// TIA Portal V17 program export: 3 tag tables, 8 data types, 18 data blocks, 27 code blocks (in call order from the OBs), 10 instance data blocks

VAR_GLOBAL   // PLC tag table "Customer"
   "VB3-M8301 Start" AT %I200.0 : Bool;   // Anfrage starten 1 = Wärmepumpe starten, 0 = nichts tun
   "VB3-M8301 Stop" AT %I200.1 : Bool;   // Stopp-Anfrage 1 = stoppen, 0 = nichts tun (überschreibt das Startsignal)
   "VB3-M8301 Freigabe" AT %I200.2 : Bool;   // Freigabe 1 = Startbefehl aktivieren 0 = Startbefehl ignorieren
   "VB3-M8301 Reset" AT %I200.3 : Bool;   // Alarmbestätigung 1 = alle Alarme löschen, 0 = nichts tun
   "VB3-M8301 Not-Aus" AT %I200.4 : Bool;   // Not-Aus zurücksetzen 1 = Not-Aus zurücksetzen, 0 = nichts tun
   "VB3-M8301 Sstop" AT %I200.5 : Bool;   // Schnellstopp-Anfrage 1 = Schnellstoppanforderung, 0 = nichts tun
   "A1024.6" AT %I200.6 : Bool;   // Reserve
   "A1024.7" AT %I200.7 : Bool;   // Reserve
   QI117_828B2 AT %I203.0 : Bool;   // Rückmeldung zur Raumlüftung WP1 1 = Lüftung ok, 0 = Startbefehl ignorieren
   QI117_828B3 AT %I203.1 : Bool;   // Kondensierbare Gase erkannt WP1 1 = Anforderung stoppen und Absperrventile schließen, 0 = nichts tun
   "A1027.2" AT %I203.2 : Bool;   // Reserve
   "A1027.3" AT %I203.3 : Bool;   // Reserve
   "A1027.4" AT %I203.4 : Bool;   // Reserve
   "A1027.5" AT %I203.5 : Bool;   // Reserve
   "A1027.6" AT %I203.6 : Bool;   // Reserve
   "VB3-M8301 Live bit" AT %I203.7 : Bool;   // Live bit
   QI117_828B1 AT %IW201 : Int;   // [%] Leistungssollwert WP1 Sollwert für die Systemleistung
   AW1028 AT %IW204 : Int;   // Reserve
   AW1030 AT %IW206 : Int;   // Reserve
   "VB3-M8301 NA-Status" AT %Q200.0 : Bool;   // Not-Aus-Status 1 = Not-Aus ok, 0 = Not-Aus aktiv
   "VB3-M8301 G1 Ein" AT %Q200.1 : Bool;   // Status der Ölheizungen Gruppe 1 1 = Heizungen ein, 0 = Heizungen aus
   "VB3-M8301 G2 Ein" AT %Q200.2 : Bool;   // Status der Ölheizungen Gruppe 2 1 = Heizungen ein, 0 = Heizungen aus
   "E1024.3" AT %Q200.3 : Bool;   // Reserve
   "E1024.4" AT %Q200.4 : Bool;   // Reserve
   "E1024.5" AT %Q200.5 : Bool;   // Reserve
   "E1024.6" AT %Q200.6 : Bool;   // Reserve
   "E1024.7" AT %Q200.7 : Bool;   // Reserve
   GH117_827 AT %Q201.0 : Bool;   // Absalzventil 1 = offen, 0 = geschlossen, gesteuert durch Heaten
   GH117_826_1 AT %Q201.1 : Bool;   // Ventil nicht kondensierbares Gase 1 1 = offen, 0 = geschlossen, gesteuert durch Heaten
   GH117_826_2 AT %Q201.2 : Bool;   // Ventil nicht kondensierbares Gase 2 1 = offen, 0 = geschlossen, gesteuert durch Heaten
   "E1025.3" AT %Q201.3 : Bool;   // Reserve
   "E1025.4" AT %Q201.4 : Bool;   // Reserve
   "E1025.5" AT %Q201.5 : Bool;   // Reserve
   "E1025.6" AT %Q201.6 : Bool;   // Reserve
   "E1025.7 Live Bit" AT %Q201.7 : Bool;   // Live bit
   "VB3-M8301 Status" AT %QW202 : Int;   // Maschinenzustand 0 = Initialisierung, 1 = Offline, 2 = Standby, Aufwärmen, Betrieb usw. (Aufzählungstyp)
   QI117_828B4 AT %QW204 : Int;   // [h] Betriebsstunden Zählt, solange der Heatbooster eingeschaltet ist
   QI117_828B5 AT %QW206 : Int;   // [h] Aktive Zeit Stunden Aktiv bedeutet, dass die Maschine eingeschaltet ist (entweder im Betrieb oder im Leerlauf).
   QI117_828B6 AT %QW208 : Int;   // [h] Laufzeit Stunden Laufen bedeutet in Betrieb (Wärmeerhöhung!)
   QI117_828B7 AT %QW210 : Int;   // [C] HBL-TT-07 (HBL-TT-901) Temperatur Saugseite Kondensator
   QI117_828B8 AT %QW212 : Int;   // [C] HBL-TT-08 (HBL-TT-518) Temperatur Druckseit Kondensator
   QI117_828B9 AT %QW214 : Int;   // [C] HBL-TT-13 (HBL-TT-546) Temperatur Saugseite Verdampfer
   QI117_828B10 AT %QW216 : Int;   // [C] HBL-TT-14 (HBL-TT-542) Temperatur Druckseit Verdampfer
   QI117_828B11 AT %QW218 : Int;   // [C] HBL-TT-16 Lufttemperatur des Containers
   QI117_828B12 AT %QW220 : Int;   // [C] HBL-TT-17 Lufttemperatur im Schaltschrank
   QI117_828B13 AT %QW222 : Int;   // [C] HBL-TT-18 Umgebungslufttemperatur
   QI117_828B16 AT %QW224 : Int;   // [ppm] HBL-CT-03 Gasdetektor Container
   QI117_828B17 AT %QW226 : Int;   // [%] SSC-LT-01 Füllstand des Sperrflüssigkeitsbehälters
   "VB3-M8301 Wärme" AT %QW228 : Int;   // [kW] Voraussichtliche Wärmelieferung
   QI117_828B18 AT %QW230 : Int;   // [1] System: COP
   "VB3-M8301 kW" AT %QW232 : Int;   // [kW] System: electrical power
   QI117_828B19 AT %QW234 : Int;   // [C] System: temperature lift
   GH117_812 AT %QW236 : Int;   // [%] Kondensatventil Verdampfer ein
   GH117_818 AT %QW238 : Int;   // [%] Dampfventil Verdampfer aus (HBL-HCV-514)
   GH117_815 AT %QW240 : Int;   // [%] Dampfventil Kondensator ein (HBL-HCV-548)
   GH117_821 AT %QW242 : Int;   // [%] Kondensatventil Kondensator aus
   EW1072 AT %QW248 : Int;   // Reserve
   "VB3-M8301 kW(1)" AT %QW244 : Int;   // Elektrische Leistung
   EW1070 AT %QW246 : Int;   // Reserve
   EW1074 AT %QW250 : Int;   // Reserve
END_VAR

VAR_GLOBAL   // PLC tag table "Default tag table"
   Clock_Byte AT %MB0 : Byte;
   Clock_10Hz AT %M0.0 : Bool;
   Clock_5Hz AT %M0.1 : Bool;
   "Clock_2.5Hz" AT %M0.2 : Bool;
   Clock_2Hz AT %M0.3 : Bool;
   "Clock_1.25Hz" AT %M0.4 : Bool;
   Clock_1Hz AT %M0.5 : Bool;
   "Clock_0.625Hz" AT %M0.6 : Bool;
   "Clock_0.5Hz" AT %M0.7 : Bool;
END_VAR

VAR_GLOBAL   // PLC tag table "Local_IO"
   DQa_0 AT %Q0.0 : Bool;
   DQa_1 AT %Q0.1 : Bool;
   DQa_2 AT %Q0.2 : Bool;
   DQa_3 AT %Q0.3 : Bool;
   DQa_4 AT %Q0.4 : Bool;
   DQa_5 AT %Q0.5 : Bool;
   DQa_6 AT %Q0.6 : Bool;
   DQa_7 AT %Q0.7 : Bool;
   DQb_0 AT %Q1.0 : Bool;
   DQb_1 AT %Q1.1 : Bool;
   DIa_0 AT %I0.0 : Bool;
   DIa_1 AT %I0.1 : Bool;
   DIa_2 AT %I0.2 : Bool;
   DIa_3 AT %I0.3 : Bool;
   DIa_4 AT %I0.4 : Bool;
   DIa_5 AT %I0.5 : Bool;
   DIa_6 AT %I0.6 : Bool;
   DIa_7 AT %I0.7 : Bool;
   DIb_0 AT %I1.0 : Bool;
   DIb_1 AT %I1.1 : Bool;
   DIb_2 AT %I1.2 : Bool;
   DIb_3 AT %I1.3 : Bool;
   DIb_4 AT %I1.4 : Bool;
   DIb_5 AT %I1.5 : Bool;
END_VAR

TYPE "stAnalogInput"
// stored: IsFailsafeCompliant false
   STRUCT
      Raw : "stRawValue";   // Raw values
      Eng : "stCalcValue";   // Engineering values
      bInitCmd : Bool;   // Recalculate scaling parameters
   END_STRUCT;
END_TYPE

TYPE "stAnalogOutput"
// stored: IsFailsafeCompliant false
   STRUCT
      Raw : "stRawValue";
      Eng { S7_SetPoint := 'True'} : "stCalcValue";
   END_STRUCT;
END_TYPE

TYPE "stCalcValue"
// stored: IsFailsafeCompliant false
   STRUCT
      fMin : Real;   // Negative-most value
      fMax : Real;   // Positive-most value
      fValue : Real;   // Actual value
      bError : Bool;   // Value invalid or out of range
      bCheckLimits : Bool := false;   // 1 = set bError if outside min & max, 0 = do nothing
      bLimited : Bool;   // 1 = value is limited, 0 = value is not limited
   END_STRUCT;
END_TYPE

TYPE "stHeartbeatCount2"
// stored: IsFailsafeCompliant false
   STRUCT
      nLocalCount : UInt;   // Count sent to remote partner
      nRemoteCount : UInt;   // Count received from remote partner
      bEnable : Bool;   // 1 = run heartbeat, 0 = disabled
      bOk : Bool;   // 1 = heatbeat ok, 0 = timeout
      nState : USInt;   // 0 = idle, 1 = ping, 2 = wait for pong, 3 = timeout
      tTimeout : Time := T#2s;   // Comm error timeout
   END_STRUCT;
END_TYPE

TYPE "stRawValue"
// stored: IsFailsafeCompliant false
   STRUCT
      iMin : Int;   // Module output at minimum input
      iMax : Int;   // Module output at maximum input
      iValue : Int;   // Current module value
      bFault : Bool;   // 0 = valid data, 1 = invalid data
   END_STRUCT;
END_TYPE

TYPE "stRegulatingValve"
// stored: IsFailsafeCompliant false
   STRUCT
      Cmd : Struct
         bManualMode : Bool;   // 1 = Manual Mode
         fManualValue : Real;   // manual position
         fOffset : Real;   // zero position offset
         Position : "stAnalogOutput";
      END_STRUCT;
      Stat : Struct
         Position : "stAnalogInput";
      END_STRUCT;
   END_STRUCT;
END_TYPE

TYPE "typeDataPtr"
// stored: IsFailsafeCompliant false
   STRUCT
      data : Array[0..7] of Word;
   END_STRUCT;
END_TYPE

TYPE "CAN-IDs_ToSend"
// stored: IsFailsafeCompliant false
   STRUCT
      IDs : Array[0..74] of Int;
   END_STRUCT;
   // IDs[0] := 16#0201;
   // IDs[1] := 16#0202;
   // IDs[2] := 16#0203;
   // IDs[3] := 16#0204;
   // IDs[4] := 16#0205;
   // IDs[5] := 16#0206;
   // IDs[6] := 16#0207;
   // IDs[7] := 16#0210;
   // IDs[8] := 16#0220;
   // IDs[9] := 16#0221;
   // IDs[10] := 16#0222;
   // IDs[11] := 16#0223;
   // IDs[12] := 16#0224;
   // IDs[13] := 16#0240;
   // IDs[14] := 16#0241;
   // IDs[15] := 16#0242;
   // IDs[16] := 16#0243;
   // IDs[17] := 16#0501;
   // IDs[18] := 16#0244;
   // IDs[19] := 16#0245;
   // IDs[20] := 16#0246;
   // IDs[21] := 16#0250;
   // IDs[22] := 16#0251;
   // IDs[23] := 16#0252;
   // IDs[24] := 16#0253;
   // IDs[25] := 16#0254;
   // IDs[26] := 16#0260;
   // IDs[27] := 16#0261;
   // IDs[28] := 16#0262;
   // IDs[29] := 16#0263;
   // IDs[30] := 16#0264;
   // IDs[31] := 16#0301;
   // IDs[32] := 16#0302;
   // IDs[33] := 16#0310;
   // IDs[34] := 16#0311;
   // IDs[35] := 16#0312;
   // IDs[36] := 16#0313;
   // IDs[37] := 16#0314;
   // IDs[38] := 16#0320;
   // IDs[39] := 16#0321;
   // IDs[40] := 16#0322;
   // IDs[41] := 16#0323;
   // IDs[42] := 16#0324;
   // IDs[43] := 16#0241;
   // IDs[44] := 16#0243;
   // IDs[45] := 16#0501;
   // IDs[46] := 16#0401;
   // IDs[47] := 16#0402;
   // IDs[48] := 16#0403;
   // IDs[49] := 16#0404;
   // IDs[50] := 16#0405;
   // IDs[51] := 16#0451;
   // IDs[52] := 16#0452;
   // IDs[53] := 16#0453;
   // IDs[54] := 16#0454;
   // IDs[55] := 16#0455;
   // IDs[56] := 16#0456;
   // IDs[57] := 16#0457;
   // IDs[58] := 16#0458;
   // IDs[59] := 16#0459;
   // IDs[60] := 16#0460;
END_TYPE

DATA_BLOCK "DB_AI"   // DB40
{ S7_Optimized_Access := 'FALSE' }
AUTHOR : Heaten
VERSION : 0.1
// stored: AutoNumber true, DBAccessibleFromOPCUA true, IsOnlyStoredInLoadMemory false, IsWriteProtectedInAS false
   VAR RETAIN
      Dummy : Bool;   // All locally-connected AIs go here
   END_VAR
BEGIN
END_DATA_BLOCK

DATA_BLOCK "DB_Calc"   // DB45
{ S7_Optimized_Access := 'FALSE' }
VERSION : 0.1
// stored: AutoNumber true, DBAccessibleFromOPCUA true, IsOnlyStoredInLoadMemory false, IsWriteProtectedInAS false
   VAR
      Dummy : Bool;   // Locally calculated values go here
   END_VAR
BEGIN
END_DATA_BLOCK

DATA_BLOCK "DB_CurrentSetting"   // DB21
{ S7_Optimized_Access := 'TRUE' }
AUTHOR : Heaten
VERSION : 0.1
// stored: AutoNumber false, DBAccessibleFromOPCUA true, IsOnlyStoredInLoadMemory false, IsRetainMemResEnabled false, IsWriteProtectedInAS false, MemoryReserve 0
   VAR RETAIN
      HeatSourceFlowLimit : Real := 0.0;   // [L/s] Heat source minimum volume flow
      HeatSinkFlowLimit : Real := 0.0;   // [L/s] Heat sink minimum volume flow
      "CAN-ModuleActive" : Bool := TRUE;   // 1 = do CAN comm, 0 = skip it
   END_VAR
BEGIN
END_DATA_BLOCK

DATA_BLOCK "DB_Customer"   // DB10
{ S7_Optimized_Access := 'TRUE' }
AUTHOR : Heaten
VERSION : 0.1
// stored: AutoNumber true, DBAccessibleFromOPCUA true, IsOnlyStoredInLoadMemory false, IsRetainMemResEnabled false, IsWriteProtectedInAS false, MemoryReserve 100
   VAR
      bEnabled : Bool;   // Enable Customer interface
      Watchdog : "stHeartbeatCount2";   // Comm monitoring Customer <-> Heatbooster
      Dummy { S7_SetPoint := 'True'} : "stCalcValue";
   END_VAR
BEGIN
END_DATA_BLOCK

DATA_BLOCK "DB_DI"   // DB2
{ S7_Optimized_Access := 'TRUE' }
VERSION : 0.1
// stored: AutoNumber false, DBAccessibleFromOPCUA true, IsOnlyStoredInLoadMemory false, IsRetainMemResEnabled false, IsWriteProtectedInAS false, MemoryReserve 0
   VAR
      EXT_FS_01 : Bool;   // Flow switch heat source (local)
      EXT_FS_02 : Bool;   // Flow switch heat sink (local)
   END_VAR
BEGIN
END_DATA_BLOCK

DATA_BLOCK "DB_DO"   // DB8
{ S7_Optimized_Access := 'TRUE' }
VERSION : 0.1
// stored: AutoNumber false, DBAccessibleFromOPCUA true, IsOnlyStoredInLoadMemory false, IsRetainMemResEnabled false, IsWriteProtectedInAS false, MemoryReserve 100
   VAR
      HBL_EC_01 : Bool;
      HBL_EC_02 : Bool;
      HBL_HV_630 : Bool;
      HBL_HV_114 : Bool;
      HBL_HV_115 : Bool;
      HBL_HV_860 : Bool;
      HBL_HV_861 : Bool;
      HBL_XV_06 : Bool;
      HBL_XV_07 : Bool;
      HBL_HV_631 : Bool;
      SSC_P_01 : Bool;
      SSC_F_01 : Bool;
      SSC_P_02 : Bool;
      CPC_P_01 : Bool;
      GH117_827 : Bool;   // Blowdown valve
      GH117_826_1 : Bool;   // NCG valve 1
      GH117_826_2 : Bool;   // NCG valve 2
      HBL_LSH_62 : Bool;
      HBL_LSL_63 : Bool;
      HBL_LSH_64 : Bool;
      HBL_LSL_864 : Bool;
      HBL_LS_632 : Bool;
      HBL_LS_633 : Bool;
   END_VAR
BEGIN
END_DATA_BLOCK

DATA_BLOCK "DB_Heatbooster"   // DB19
{ S7_Optimized_Access := 'TRUE' }
VERSION : 0.1
// stored: AutoNumber true, DBAccessibleFromOPCUA true, IsOnlyStoredInLoadMemory false, IsRetainMemResEnabled false, IsWriteProtectedInAS false, MemoryReserve 0
   VAR
      AI : Struct
         HBL_TT_502 { S7_SetPoint := 'True'} : "stCalcValue";   // Compressor discharge popoff temperature
         HBL_PT_503 { S7_SetPoint := 'True'} : "stCalcValue";   // Compressor discharge pressure
         HBL_TT_504 { S7_SetPoint := 'True'} : "stCalcValue";   // Compressor discharge temperature
         HBL_LT_510 { S7_SetPoint := 'True'} : "stCalcValue";   // Steam generator condensate level
         HBL_PT_511 { S7_SetPoint := 'True'} : "stCalcValue";   // Heat sink discharge pressure
         HBL_TT_512 { S7_SetPoint := 'True'} : "stCalcValue";   // Heat sink discharge temperature
         HBL_TT_516 { S7_SetPoint := 'True'} : "stCalcValue";   // Steam generator suction temperature
         HBL_PT_517 { S7_SetPoint := 'True'} : "stCalcValue";   // Steam generator suction pressure
         HBL_TT_518 { S7_SetPoint := 'True'} : "stCalcValue";   // Heat sink discharge process temperature
         HBL_PT_519 { S7_SetPoint := 'True'} : "stCalcValue";   // Heat sink discharge process pressure
         HBL_FT_520 { S7_SetPoint := 'True'} : "stCalcValue";   // Refrigerant flow
         HBL_TT_530 { S7_SetPoint := 'True'} : "stCalcValue";   // Expansion valve B discharge temperature
         HBL_PT_531 { S7_SetPoint := 'True'} : "stCalcValue";   // Expansion valve B discharge pressure
         HBL_TT_532 { S7_SetPoint := 'True'} : "stCalcValue";   // Heat source discharge B temperature
         HBL_TT_533 { S7_SetPoint := 'True'} : "stCalcValue";   // Evaporator B discharge temperature
         HBL_PT_534 { S7_SetPoint := 'True'} : "stCalcValue";   // Evaporator B discharge pressure
         HBL_AT_535 { S7_SetPoint := 'True'} : "stCalcValue";   // Evaporator B steam quality
         HBL_TT_540 { S7_SetPoint := 'True'} : "stCalcValue";   // Expansion valve A discharge temperature
         HBL_PT_541 { S7_SetPoint := 'True'} : "stCalcValue";   // Expansion valve A discharge pressure
         HBL_TT_542 { S7_SetPoint := 'True'} : "stCalcValue";   // Heat source discharge temperature
         HBL_TT_543 { S7_SetPoint := 'True'} : "stCalcValue";   // Evaporator A discharge temperature
         HBL_PT_544 { S7_SetPoint := 'True'} : "stCalcValue";   // Evaporator A discharge pressure
         HBL_AT_545 { S7_SetPoint := 'True'} : "stCalcValue";   // Evaporator A steam quality
         HBL_TT_546 { S7_SetPoint := 'True'} : "stCalcValue";   // Heat source suction temperature
         HBL_PT_547 { S7_SetPoint := 'True'} : "stCalcValue";   // Heast source suction pressure
         HBL_TT_571 { S7_SetPoint := 'True'} : "stCalcValue";   // Compressor suction temperature
         HBL_PT_572 { S7_SetPoint := 'True'} : "stCalcValue";   // Compressor suction pressure
         HBL_TT_573 { S7_SetPoint := 'True'} : "stCalcValue";   // Expansion valve suction temperature
         HBL_LT_610 { S7_SetPoint := 'True'} : "stCalcValue";   // HP receiver refrigerant level
         HBL_TT_611 { S7_SetPoint := 'True'} : "stCalcValue";   // Steam generator discharge temperature
         HBL_PT_612 { S7_SetPoint := 'True'} : "stCalcValue";   // Steam generator discharge pressure
         HBL_CT_615 { S7_SetPoint := 'True'} : "stCalcValue";   // Gas detector PSV discharge pipe
         HBL_PT_618 { S7_SetPoint := 'True'} : "stCalcValue";   // HP Receiver pressure
         HBL_PT_635 { S7_SetPoint := 'True'} : "stCalcValue";   // Oil separator stage 1 oil return pressure
         HBL_PT_636 { S7_SetPoint := 'True'} : "stCalcValue";   // Oil separator stage 2 oil return pressure
         HBL_LT_650 { S7_SetPoint := 'True'} : "stCalcValue";   // Heat source condensate buffer tank level
         HBL_PT_651 { S7_SetPoint := 'True'} : "stCalcValue";   // Heat source condensate buffer tank pressure
         HBL_PT_701 { S7_SetPoint := 'True'} : "stCalcValue";   // Filter dryer suction pressure
         HBL_PT_702 { S7_SetPoint := 'True'} : "stCalcValue";   // Filter dryer discharge pressure
         HBL_PT_703 { S7_SetPoint := 'True'} : "stCalcValue";   // Filter dryer differential pressure
         CPC_LT_870 { S7_SetPoint := 'True'} : "stCalcValue";   // CPC tank refrigerant level
         CPC_TT_871 { S7_SetPoint := 'True'} : "stCalcValue";   // CPC tank refrigerant temperature
         CPC_PT_872 { S7_SetPoint := 'True'} : "stCalcValue";   // CPC tank refrigerant pressure
         CPC_PT_862 { S7_SetPoint := 'True'} : "stCalcValue";   // CPC pump discharge pressure
         HBL_TT_901 { S7_SetPoint := 'True'} : "stCalcValue";   // Heat sink suction temperature
         HBL_PT_902 { S7_SetPoint := 'True'} : "stCalcValue";   // Heat sink suction pressure
         HBL_TT_03 { S7_SetPoint := 'True'} : "stCalcValue";   // Oil sump oil temperature
         HBL_TT_16 { S7_SetPoint := 'True'} : "stCalcValue";   // Container air temperature
         HBL_TT_17 { S7_SetPoint := 'True'} : "stCalcValue";   // Control cabinet air temperature
         HBL_TT_18 { S7_SetPoint := 'True'} : "stCalcValue";   // Ambient air temperature
         HBL_TT_20 { S7_SetPoint := 'True'} : "stCalcValue";   // Compressor motor winding temperature
         HBL_TT_21 { S7_SetPoint := 'True'} : "stCalcValue";   // Oil sump wall temperature left
         HBL_TT_22 { S7_SetPoint := 'True'} : "stCalcValue";   // Oil sump wall temperature right
         HBL_TT_23 { S7_SetPoint := 'True'} : "stCalcValue";   // Compressor motor U-winding temperature
         HBL_TT_24 { S7_SetPoint := 'True'} : "stCalcValue";   // Compressor motor V-winding temperature
         HBL_TT_25 { S7_SetPoint := 'True'} : "stCalcValue";   // Compressor motor W-winding temperature
         HBL_TT_26 { S7_SetPoint := 'True'} : "stCalcValue";   // Compressor motor D bearing temperature
         HBL_TT_27 { S7_SetPoint := 'True'} : "stCalcValue";   // Compressor motor N bearing temperature
         HBL_PT_05 { S7_SetPoint := 'True'} : "stCalcValue";   // Crankcase gas pressure
         HBL_PT_06 { S7_SetPoint := 'True'} : "stCalcValue";   // Oil pump discharge pressure
         HBL_PT_17 { S7_SetPoint := 'True'} : "stCalcValue";   // Oil gallery pressure
         HBL_CT_01 { S7_SetPoint := 'True'} : "stCalcValue";   // Gas detector Heatbooster (optional)
         HBL_CT_03 { S7_SetPoint := 'True'} : "stCalcValue";   // Gas detector container (optional)
         SSC_TT_01 { S7_SetPoint := 'True'} : "stCalcValue";   // SSC seal suction temperature
         SSC_TT_02 { S7_SetPoint := 'True'} : "stCalcValue";   // SSC seal discharge temperature
         SSC_TT_03 { S7_SetPoint := 'True'} : "stCalcValue";   // SSC barrier fluid circulation pump suction temperature
         SSC_TT_04 { S7_SetPoint := 'True'} : "stCalcValue";   // SSC barrier fluid heat exchanger temperature
         SSC_PIT_01 { S7_SetPoint := 'True'} : "stCalcValue";   // SSC barrier fluid accumulator pressure
         SSC_PDT_01 { S7_SetPoint := 'True'} : "stCalcValue";   // SSC barrier fluid circulation pump differential pressure
         SSC_LT_01 { S7_SetPoint := 'True'} : "stCalcValue";   // SSC barrier fluid reservoir level
         HBL_VT_01 { S7_SetPoint := 'True'} : "stCalcValue";   // [?] Oil sump oil viscosity
         HBL_TT_36 { S7_SetPoint := 'True'} : "stCalcValue";   // [C] Oil sump oil viscosity probe temperature
      END_STRUCT;
      Calc : Struct
         Compressor : Struct
            CrankcaseSaturationTemperature { S7_SetPoint := 'True'} : "stCalcValue";   // C
            CrankcaseSuperheat { S7_SetPoint := 'True'} : "stCalcValue";   // C
            VolumetricEfficiency { S7_SetPoint := 'True'} : "stCalcValue";   // %
            IsentropicEfficiency { S7_SetPoint := 'True'} : "stCalcValue";   // %
            Massflow { S7_SetPoint := 'True'} : "stCalcValue";   // kg/h
         END_STRUCT;
         HeatSink : Struct
            DeltaT { S7_SetPoint := 'True'} : "stCalcValue";
            Pinch { S7_SetPoint := 'True'} : "stCalcValue";
            HeatRate { S7_SetPoint := 'True'} : "stCalcValue";
            DeltaP { S7_SetPoint := 'True'} : "stCalcValue";
            Massflow { S7_SetPoint := 'True'} : "stCalcValue";
         END_STRUCT;
         HeatSource : Struct
            DeltaT { S7_SetPoint := 'True'} : "stCalcValue";
            Pinch { S7_SetPoint := 'True'} : "stCalcValue";
            HeatRate { S7_SetPoint := 'True'} : "stCalcValue";
            DeltaP { S7_SetPoint := 'True'} : "stCalcValue";
            TemperatureRateOfChange { S7_SetPoint := 'True'} : "stCalcValue";
            Massflow { S7_SetPoint := 'True'} : "stCalcValue";
         END_STRUCT;
         HighPressPart : Struct
            CompressorSaturationTemperature { S7_SetPoint := 'True'} : "stCalcValue";
            CompressorSuperheat { S7_SetPoint := 'True'} : "stCalcValue";
            CondenserSaturationTemperature { S7_SetPoint := 'True'} : "stCalcValue";
            CondenserSubcooling { S7_SetPoint := 'True'} : "stCalcValue";
            ExpansionValveSubcooling { S7_SetPoint := 'True'} : "stCalcValue";
            CondenserDeltaP { S7_SetPoint := 'True'} : "stCalcValue";
         END_STRUCT;
         LowPressPart : Struct
            EvaporatorSuperheat { S7_SetPoint := 'True'} : "stCalcValue";
            CompressorSuperheat { S7_SetPoint := 'True'} : "stCalcValue";
            EvaporatorSaturationTemperature { S7_SetPoint := 'True'} : "stCalcValue";
            CompressorSaturationTemperature { S7_SetPoint := 'True'} : "stCalcValue";
         END_STRUCT;
         System : Struct
            Quality { S7_SetPoint := 'True'} : "stCalcValue";
            COP { S7_SetPoint := 'True'} : "stCalcValue";
            ElectricalPower { S7_SetPoint := 'True'} : "stCalcValue";
            TemperatureLift { S7_SetPoint := 'True'} : "stCalcValue";
            MotorEfficiency { S7_SetPoint := 'True'} : "stCalcValue";
            FMEP { S7_SetPoint := 'True'} : "stCalcValue";
         END_STRUCT;
         Auxiliary : Struct
            ShaftSealDeltaT { S7_SetPoint := 'True'} : "stCalcValue";
            CPCPumpDeltaP { S7_SetPoint := 'True'} : "stCalcValue";
         END_STRUCT;
         Misc : Struct
            EvaporatorDischargePressureMean { S7_SetPoint := 'True'} : "stCalcValue";
            EvaporatorDischargeTemperatureMin { S7_SetPoint := 'True'} : "stCalcValue";
            EvaporatorDischargeTemperatureMean { S7_SetPoint := 'True'} : "stCalcValue";
            OilFilterDeltaP { S7_SetPoint := 'True'} : "stCalcValue";
         END_STRUCT;
      END_STRUCT;
      DI : Struct
         HBL_FS_01 : Bool;
         HBL_FS_02 : Bool;
         HBL_LS_632 : Bool;
         HBL_LS_633 : Bool;
         CPC_LS_864 : Bool;
         VPNUserConnected : Bool;
      END_STRUCT;
      "DO" : Struct
         HBL_EC_01 : Bool;
         HBL_EC_02 : Bool;
         HBL_HV_630 : Bool;
         HBL_HV_114 : Bool;
         HBL_HV_115 : Bool;
         HBL_HV_860 : Bool;
         HBL_HV_861 : Bool;
         SSC_P_01 : Bool;
         SSC_F_01 : Bool;
         SSC_P_02 : Bool;
         CPC_P_01 : Bool;
         SpareContactor1 : Bool;
         SpareContactor2 : Bool;
         HBL_HV_631 : Bool;
      END_STRUCT;
      Inverter : Struct
         HBL_SC_01_A1 { S7_SetPoint := 'True'} : "stCalcValue";   // Container ventilation fan speed
         HBL_SC_01_A2 { S7_SetPoint := 'True'} : "stCalcValue";   // Container ventilation fan torque
         HBL_SC_01_A3 { S7_SetPoint := 'True'} : "stCalcValue";   // Container ventilation fan power
         HBL_SC_02_A1 { S7_SetPoint := 'True'} : "stCalcValue";   // Compressor lubrication pump speed
         HBL_SC_02_A2 { S7_SetPoint := 'True'} : "stCalcValue";   // Compressor lubrication pump torque
         HBL_SC_02_A3 { S7_SetPoint := 'True'} : "stCalcValue";   // Compressor lubrication pump power
         HBL_SC_03_A1 { S7_SetPoint := 'True'} : "stCalcValue";   // CPC pump speed
         HBL_SC_03_A2 { S7_SetPoint := 'True'} : "stCalcValue";   // CPC pump torque
         HBL_SC_03_A3 { S7_SetPoint := 'True'} : "stCalcValue";   // CPC pump power
         HBL_SC_10_A1 { S7_SetPoint := 'True'} : "stCalcValue";   // Compressor motor speed
         HBL_SC_10_A2 { S7_SetPoint := 'True'} : "stCalcValue";   // Compressor motor torque
         HBL_SC_10_A3 { S7_SetPoint := 'True'} : "stCalcValue";   // Compressor motor power
      END_STRUCT;
      Valve : Struct
         HBL_HCV_576_A1 : "stCalcValue";   // Expansion Valve A
         HBL_HCV_578_A1 : "stCalcValue";   // Expansion Valve B
         HBL_HCV_577_A1 { S7_SetPoint := 'True'} : "stCalcValue";   // Expansion Valve A2
         HBL_HCV_579_A1 { S7_SetPoint := 'True'} : "stCalcValue";   // Expansion Valve B2
         HBL_HCV_515_A1 { S7_SetPoint := 'True'} : "stCalcValue";   // Heat sink condensate blowdown flow control valve
         HBL_HCV_575_A1 { S7_SetPoint := 'True'} : "stCalcValue";   // Recuperator oil drain valve
         HBL_HCV_616_A1 { S7_SetPoint := 'True'} : "stCalcValue";   // Recuperator bypass valve
         HBL_HCV_700_A1 { S7_SetPoint := 'True'} : "stCalcValue";   // Oil recovery refrigerant blowdown valve
         HBL_HCV_514_A1 { S7_SetPoint := 'True'} : "stCalcValue";   // Heat sink discharge pressure control valve
         HBL_HCV_548_A1 { S7_SetPoint := 'True'} : "stCalcValue";   // Heat source suction pressure control valve
      END_STRUCT;
   END_VAR
BEGIN
END_DATA_BLOCK

DATA_BLOCK "DB_InverterDrives"   // DB41
{ S7_Optimized_Access := 'FALSE' }
VERSION : 0.1
// stored: AutoNumber false, DBAccessibleFromOPCUA true, IsOnlyStoredInLoadMemory false, IsWriteProtectedInAS false
   VAR
      Dummy : Bool;   // Locally-connected inverters go here
   END_VAR
BEGIN
END_DATA_BLOCK

DATA_BLOCK "DB_System"   // DB42
{ S7_Optimized_Access := 'TRUE' }
VERSION : 0.1
// stored: AutoNumber false, DBAccessibleFromOPCUA true, IsOnlyStoredInLoadMemory false, IsRetainMemResEnabled false, IsWriteProtectedInAS false, MemoryReserve 100
   VAR
      bFirstCycle : Bool := FALSE;   // High on first scan only
      bFirstCycleCyclic : Bool := FALSE;
      bSimulation : Bool := FALSE;   // Simulation active
      SoftwareVersion : String := 'V4.0.0.7';   // PLC software version string
      S7CommEnable : Bool := true;   // Do S7 comm with Process PLC
   END_VAR
   VAR RETAIN
      ClientID : String := 'default';   // used by MQTT
   END_VAR
BEGIN
END_DATA_BLOCK

DATA_BLOCK "DB_TestSupport"   // DB6
{ S7_Optimized_Access := 'TRUE' }
VERSION : 0.1
// stored: AutoNumber true, DBAccessibleFromOPCUA true, IsOnlyStoredInLoadMemory false, IsRetainMemResEnabled false, IsWriteProtectedInAS false, MemoryReserve 100
   VAR
      AI : Struct
         TSS_TT_201 { S7_SetPoint := 'True'} : "stCalcValue";   // Heat source tank temperature
         TSS_TT_202 { S7_SetPoint := 'True'} : "stCalcValue";   // Heat sink tank temperature
         TSS_TT_206 { S7_SetPoint := 'True'} : "stCalcValue";   // Heat source suction temperature
         TSS_TT_208 { S7_SetPoint := 'True'} : "stCalcValue";   // Heat sink suction temperature
         TSS_TT_209 { S7_SetPoint := 'True'} : "stCalcValue";   // Heat sink discharge temperature
         TSS_FT_210 { S7_SetPoint := 'True'} : "stCalcValue";   // Heat source flow
         TSS_FT_211 { S7_SetPoint := 'True'} : "stCalcValue";   // Heat sink flow
         TSS_SC_213 { S7_SetPoint := 'True'} : "stCalcValue";   // Heat source feed pump speed
         TSS_SC_214 { S7_SetPoint := 'True'} : "stCalcValue";   // Heat sink feed pump speed
         TSA_PT_300 { S7_SetPoint := 'True'} : "stCalcValue";   // Heat sink cycle condensate pump suction pressure
         TSA_TT_301 { S7_SetPoint := 'True'} : "stCalcValue";   // Heat sink cycle condensate pump suction temperature
         TSA_TT_304 { S7_SetPoint := 'True'} : "stCalcValue";   // Heat sink cycle condensate tank suction temperature
         TSA_PT_306 { S7_SetPoint := 'True'} : "stCalcValue";   // Heat sink cycle condensate pump discharge pressure
         TSA_FT_307 { S7_SetPoint := 'True'} : "stCalcValue";   // Heat sink cycle condensate pump discharge flow
         TSA_LT_308 { S7_SetPoint := 'True'} : "stCalcValue";   // Heat sink cycle condensate tank level
         TSA_TT_320 { S7_SetPoint := 'True'} : "stCalcValue";   // Steam generator discharge temperature
         TSA_PT_321 { S7_SetPoint := 'True'} : "stCalcValue";   // Steam generator discharge pressure
         TSA_PT_323 { S7_SetPoint := 'True'} : "stCalcValue";   // Steam system pressure (?)
         TSA_TT_324 { S7_SetPoint := 'True'} : "stCalcValue";   // Steam system temperature (?)
         TSA_PT_328 { S7_SetPoint := 'True'} : "stCalcValue";   // Nitrogen blanketing pressure
         TSA_PT_350 { S7_SetPoint := 'True'} : "stCalcValue";   // Heat source cycle condensate pump suction pressure
         TSA_TT_351 { S7_SetPoint := 'True'} : "stCalcValue";   // Heat source cycle condensate pump suction temperature
         TSA_PT_354 { S7_SetPoint := 'True'} : "stCalcValue";   // Heat source cycle condensate pump discharge pressure
         TSA_FT_355 { S7_SetPoint := 'True'} : "stCalcValue";   // Heat source cycle condensate pump discharge flow
         TSA_TT_356 { S7_SetPoint := 'True'} : "stCalcValue";   // Heat source suction temperature
         TSA_PT_374 { S7_SetPoint := 'True'} : "stCalcValue";   // Heat source suction pressure
      END_STRUCT;
      DI : Struct
         TSA_HV_326 : Bool;   // Heat sink cycle nitrogen blanketing valve 1
         TSA_HV_327 : Bool;   // Heat sink cycle nitrogen blanketing valve 2
         TSA_HV_330 : Bool;   // Preheating pump discharge valve
         TSA_HV_372 : Bool;   // Heat source cycle nitrogen blanketing valve 1
         TSA_HV_373 : Bool;   // Heat source cycle nitrogen blanketing valve 2
         Spare05 : Bool;
         Spare06 : Bool;
         Spare07 : Bool;
         Spare10 : Bool;
         Spare11 : Bool;
         Spare12 : Bool;
         Spare13 : Bool;
         Spare14 : Bool;
         Spare15 : Bool;
         Spare16 : Bool;
         Spare17 : Bool;
      END_STRUCT;
      Valve : Struct
         TSS_HCV_301_A1 { S7_SetPoint := 'True'} : "stCalcValue";   // Heat source 3-way mix valve position
         TSS_HCV_302_A1 { S7_SetPoint := 'True'} : "stCalcValue";   // Heat sink 3-way mix valve position
         TSA_HCV_322_A1 { S7_SetPoint := 'True'} : "stCalcValue";   // Heat sink cycle control valve position
         TSA_HCV_370_A1 { S7_SetPoint := 'True'} : "stCalcValue";   // Heat source cycle control valve position
      END_STRUCT;
      Inverter : Struct
         TSA_SC_301 : "stCalcValue";
         TSA_SC_330 : "stCalcValue";
         TSA_SC_351 : "stCalcValue";
      END_STRUCT;
   END_VAR
BEGIN
END_DATA_BLOCK

DATA_BLOCK "DB_Valves"   // DB46
{ S7_Optimized_Access := 'FALSE' }
AUTHOR : Heaten
VERSION : 0.1
// stored: AutoNumber false, DBAccessibleFromOPCUA true, IsOnlyStoredInLoadMemory false, IsWriteProtectedInAS false
   VAR RETAIN
      GH117_815 { S7_SetPoint := 'True'} : "stRegulatingValve";   // Dampfventil Kondensator ein
      GH117_821 { S7_SetPoint := 'True'} : "stRegulatingValve";   // Kondensatventil Kondensator aus
      GH117_812 { S7_SetPoint := 'True'} : "stRegulatingValve";   // Kondensatventil Verdampfer ein
      GH117_818 { S7_SetPoint := 'True'} : "stRegulatingValve";   // Dampfventil Verdampfer aus
   END_VAR
BEGIN
   GH117_815.Cmd.Position.Raw.iMin := 0;
   GH117_815.Cmd.Position.Raw.iMax := 1000;
   GH117_815.Cmd.Position.Eng.fMin := 0.0;
   GH117_815.Cmd.Position.Eng.fMax := 100.0;
   GH117_821.Cmd.Position.Raw.iMin := 0;
   GH117_821.Cmd.Position.Raw.iMax := 1000;
   GH117_821.Cmd.Position.Eng.fMin := 0.0;
   GH117_821.Cmd.Position.Eng.fMax := 100.0;
   GH117_812.Cmd.Position.Raw.iMin := 0;
   GH117_812.Cmd.Position.Raw.iMax := 1000;
   GH117_812.Cmd.Position.Eng.fMin := 0.0;
   GH117_812.Cmd.Position.Eng.fMax := 100.0;
   GH117_818.Cmd.Position.Raw.iMin := 0;
   GH117_818.Cmd.Position.Raw.iMax := 1000;
   GH117_818.Cmd.Position.Eng.fMin := 0.0;
   GH117_818.Cmd.Position.Eng.fMax := 100.0;
END_DATA_BLOCK

DATA_BLOCK "DB_Cloud"   // DB200
{ S7_Optimized_Access := 'TRUE' }
VERSION : 0.1
// stored: AutoNumber false, DBAccessibleFromOPCUA true, IsOnlyStoredInLoadMemory false, IsRetainMemResEnabled false, IsWriteProtectedInAS false, MemoryReserve 0
   VAR
      HBL_TT_502 : Real;
      HBL_PT_503 : Real;
      HBL_TT_504 : Real;
      HBL_LT_510 : Real;
      HBL_PT_511 : Real;
      HBL_TT_512 : Real;
      HBL_TT_516 : Real;
      HBL_PT_517 : Real;
      HBL_TT_518 : Real;
      HBL_PT_519 : Real;
      HBL_FT_520 : Real;
      HBL_TT_530 : Real;
      HBL_PT_531 : Real;
      HBL_TT_532 : Real;
      HBL_TT_533 : Real;
      HBL_PT_534 : Real;
      HBL_AT_535 : Real;
      HBL_TT_540 : Real;
      HBL_PT_541 : Real;
      HBL_TT_542 : Real;
      HBL_TT_543 : Real;
      HBL_PT_544 : Real;
      HBL_AT_545 : Real;
      HBL_TT_546 : Real;
      HBL_PT_547 : Real;
      HBL_TT_571 : Real;
      HBL_PT_572 : Real;
      HBL_TT_573 : Real;
      HBL_LT_610 : Real;
      HBL_TT_611 : Real;
      HBL_PT_612 : Real;
      HBL_CT_615 : Real;
      HBL_PT_618 : Real;
      HBL_PT_635 : Real;
      HBL_PT_636 : Real;
      HBL_LT_650 : Real;
      HBL_PT_651 : Real;
      HBL_PT_701 : Real;
      HBL_PT_702 : Real;
      HBL_PT_703 : Real;
      CPC_LT_870 : Real;
      CPC_TT_871 : Real;
      CPC_PT_872 : Real;
      CPC_PT_862 : Real;
      HBL_TT_901 : Real;
      HBL_PT_902 : Real;
      HBL_TT_03 : Real;
      HBL_TT_16 : Real;
      HBL_TT_17 : Real;
      HBL_TT_18 : Real;
      HBL_TT_20 : Real;
      HBL_TT_21 : Real;
      HBL_TT_22 : Real;
      HBL_TT_23 : Real;
      HBL_TT_24 : Real;
      HBL_TT_25 : Real;
      HBL_TT_26 : Real;
      HBL_TT_27 : Real;
      HBL_PT_05 : Real;
      HBL_PT_06 : Real;
      HBL_PT_17 : Real;
      HBL_CT_01 : Real;
      HBL_CT_03 : Real;
      SSC_TT_01 : Real;
      SSC_TT_02 : Real;
      SSC_TT_03 : Real;
      SSC_TT_04 : Real;
      SSC_PIT_01 : Real;
      SSC_PDT_01 : Real;
      SSC_LT_01 : Real;
      HBL_VT_01 : Real;
      HBL_TT_36 : Real;
      Compressor_CrankcaseSaturationTemperature : Real;
      Compressor_CrankcaseSuperheat : Real;
      Compressor_VolumetricEfficiency : Real;
      Compressor_IsentropicEfficiency : Real;
      Compressor_Massflow : Real;
      HeatSink_DeltaT : Real;
      HeatSink_Pinch : Real;
      HeatSink_HeatRate : Real;
      HeatSink_DeltaP : Real;
      HeatSink_Massflow : Real;
      HeatSource_DeltaT : Real;
      HeatSource_Pinch : Real;
      HeatSource_HeatRate : Real;
      HeatSource_DeltaP : Real;
      HeatSource_TemperatureRateOfChange : Real;
      HeatSource_Massflow : Real;
      HighPressPart_CompressorSaturationTemperature : Real;
      HighPressPart_CompressorSuperheat : Real;
      HighPressPart_CondenserSaturationTemperature : Real;
      HighPressPart_CondenserSubcooling : Real;
      HighPressPart_ExpansionValveSubcooling : Real;
      HighPressPart_CondenserDeltaP : Real;
      LowPressPart_EvaporatorSuperheat : Real;
      LowPressPart_CompressorSuperheat : Real;
      LowPressPart_EvaporatorSaturationTemperature : Real;
      LowPressPart_CompressorSaturationTemperature : Real;
      System_Quality : Real;
      System_COP : Real;
      System_ElectricalPower : Real;
      System_TemperatureLift : Real;
      System_MotorEfficiency : Real;
      System_FMEP : Real;
      Auxiliary_ShaftSealDeltaT : Real;
      Auxiliary_CPCPumpDeltaP : Real;
      Misc_OilFilterDeltaP : Real;
      HBL_FS_01 : Bool;
      HBL_FS_02 : Bool;
      HBL_LS_632 : Bool;
      HBL_LS_633 : Bool;
      CPC_LS_864 : Bool;
      VPNUserConnected : Bool;
      HBL_EC_01 : Bool;
      HBL_EC_02 : Bool;
      HBL_HV_630 : Bool;
      HBL_HV_860 : Bool;
      HBL_HV_861 : Bool;
      SSC_P_01 : Bool;
      SSC_F_01 : Bool;
      SSC_P_02 : Bool;
      CPC_P_01 : Bool;
      HBL_HV_631 : Bool;
      HBL_SC_01_A1 : Real;
      HBL_SC_01_A2 : Real;
      HBL_SC_01_A3 : Real;
      HBL_SC_02_A1 : Real;
      HBL_SC_02_A2 : Real;
      HBL_SC_02_A3 : Real;
      HBL_SC_03_A1 : Real;
      HBL_SC_03_A2 : Real;
      HBL_SC_03_A3 : Real;
      HBL_SC_10_A1 : Real;
      HBL_SC_10_A2 : Real;
      HBL_SC_10_A3 : Real;
      HBL_HCV_576_A1 : Real;
      HBL_HCV_578_A1 : Real;
      HBL_HCV_577_A1 : Real;
      HBL_HCV_579_A1 : Real;
      HBL_HCV_515_A1 : Real;
      HBL_HCV_575_A1 : Real;
      HBL_HCV_616_A1 : Real;
      HBL_HCV_700_A1 : Real;
      HBL_HCV_514_A1 : Real;
      HBL_HCV_548_A1 : Real;
      ClientID : String;
      RunningTimeHours : Int;
      RunningTimeMinutes : Int;
      RunningTimeSeconds : Int;
      MachineState : Int;
   END_VAR
BEGIN
END_DATA_BLOCK

DATA_BLOCK "DB_FromHB"   // DB100
{ S7_Optimized_Access := 'FALSE' }
VERSION : 0.1
// stored: AutoNumber false, DBAccessibleFromOPCUA true, IsOnlyStoredInLoadMemory false, IsWriteProtectedInAS false
   VAR
      CompressorMotorPower : Real;   // [kW]
      CompressorMotorSpeed : Real;   // [rpm]
      HBL_CT_524 : Real;   // [ppm]
      HBL_CT_538 : Real;   // [ppm]
      HBL_CT_615 : Real;   // [ppm]
      HBL_CT_620 : Real;   // [ppm]
      HBL_CT_643 : Real;   // [ppm]
      HBL_CT_673 : Real;   // [ppm]
      TemperatureLift : Real;   // [C]
      COP : Real;   // [1]
      HeatSinkHeatRate : Real;   // [kW]
      HeatboosterPerformance : Real;   // [%]
      WatchdogCounter : UInt;   // Liveness counter (free-running)
      RunningTimeHours : UInt;   // [h]
      RunningTimeMinutes : UInt;   // [min]
      RunningTimeSeconds : UInt;   // [s]
      HeatboosterState : UInt;   // 0 = Initialization, 1 = Offline, 2 = Standby, 3 = Prepare start, 4 = Start, 5 = Warmup, 6 = Run, 7 = Stop
      EmergencyStopStatus : Bool;   // 1 = E-stop ok, 0 = E-stop active
      AlarmActive : Bool;   // 1 = Common alarm active, 0 = Common alarm not active
      WarningActive : Bool;   // 1 = Common warning active, 0 = Common warning not active
      HBL_EC_01 : Bool;   // 1 = heaters on, 0 = heaters off
      HBL_EC_02 : Bool;   // 1 = heaters on, 0 = heaters off
      SSC_P_01 : Bool;   // 1 = pump running, 0 = pump off
      SSC_P_02 : Bool;   // 1 = pump running, 0 = pump off
      SSC_F_01 : Bool;   // 1 = fan running, 0 = fan off
      HBL_PZH_539 : Bool;   // 1 = switch active, 0 = switch not active
      HBL_HV_563 : Bool;
      HBL_HV_564 : Bool;
      HBL_HV_630 : Bool;
      HBL_HV_631 : Bool;
      HBL_HV_640_X1 : Bool;
      HBL_HV_640_X2 : Bool;
      HBL_HV_670_X1 : Bool;
      HBL_HV_670_X2 : Bool;
      HBL_HV_676 : Bool;
      CPC_HV_852_X1 : Bool;
      CPC_HV_852_X2 : Bool;
      HBL_HV_861_X1 : Bool;
      HBL_HV_861_X2 : Bool;
      CPC_LSH_870A : Bool;
      CPC_LSL_870B : Bool;
      CPC_PSH_874 : Bool;
      HBL_LSH_632 : Bool;
      HBL_LSL_633 : Bool;
      HBL_LS_644 : Bool;
      HBL_LS_674 : Bool;
      Spare615 : Bool;
      Spare616 : Bool;
      Spare617 : Bool;
      Alarms : Array[0..191] of Bool;   // 0 = no alarm, 1 = active or active unacknowledged alarm
      HBL_SC_03_A1 : Real;   // [rpm]
      HBL_SC_03_A2 : Real;   // [%]
      HBL_SC_03_A3 : Real;   // [kW]
      HBL_SC_01_A1 : Real;   // [rpm]
      HBL_SC_01_A2 : Real;   // [%]
      HBL_SC_01_A3 : Real;   // [kW]
      HBL_SC_02_A1 : Real;   // [rpm]
      HBL_SC_02_A2 : Real;   // [%]
      HBL_SC_02_A3 : Real;   // [kW]
      HBL_SC_10_A1 : Real;   // [rpm]
      HBL_SC_10_A2 : Real;   // [%]
      HBL_SC_10_A3 : Real;   // [kW]
      HBL_TT_18 : Real;   // [C]
      HBL_TT_03 : Real;   // [C]
      HBL_TT_21 : Real;   // [C]
      HBL_TT_22 : Real;   // [C]
      SSC_LT_01 : Real;
      SSC_PDT_01 : Real;
      SSC_PIT_01 : Real;
      SSC_TT_01 : Real;   // [C]
      SSC_TT_02 : Real;   // [C]
      SSC_TT_03 : Real;   // [C]
      SSC_TT_04 : Real;   // [C]
      HBL_TT_502 : Real;   // [C]
      HBL_PT_503 : Real;
      HBL_TT_504 : Real;   // [C]
      HBL_TT_505 : Real;   // [C]
      HBL_PT_506 : Real;
      HBL_LT_510 : Real;
      HBL_PT_511 : Real;
      HBL_TT_512 : Real;   // [C]
      HBL_HCV_514_A1 : Real;
      HBL_HCV_515_A1 : Real;
      HBL_TT_516 : Real;   // [C]
      HBL_PT_517 : Real;
      HBL_TT_518 : Real;   // [C]
      HBL_PT_519 : Real;
      HBL_TT_525 : Real;
      HBL_PT_526 : Real;
      HBL_FT_527 : Real;
      HBL_TT_530 : Real;
      HBL_PT_531 : Real;
      HBL_TT_532 : Real;
      HBL_TT_533 : Real;
      HBL_PT_534 : Real;
      HBL_AT_535 : Real;
      HBL_TT_16 : Real;
      HBL_TT_540 : Real;
      HBL_PT_541 : Real;
      HBL_TT_542 : Real;
      HBL_TT_543 : Real;
      HBL_PT_544 : Real;
      HBL_AT_545 : Real;
      HBL_TT_546 : Real;
      HBL_PT_547 : Real;
      HBL_HCV_548_A1 : Real;
      HBL_TT_17 : Real;
      HBL_PT_561 : Real;
      HBL_PT_562 : Real;
      HBL_FT_565 : Real;
      HBL_FT_566 : Real;
      HBL_TT_571 : Real;
      HBL_PT_572 : Real;
      HBL_TT_573 : Real;
      HBL_HCV_575_A1 : Real;
      HBL_HCV_576_A1 : Real;
      HBL_HCV_578_A1 : Real;
      HBL_PT_580 : Real;
      HBL_LIT_610 : Real;
      HBL_TT_611 : Real;
      HBL_PT_612 : Real;
      HBL_HCV_616_A1 : Real;
      HBL_PT_618 : Real;
      HBL_HCV_700_A1 : Real;
      HBL_PT_701 : Real;
      HBL_PT_702 : Real;
      HBL_PT_05 : Real;
      HBL_TT_23 : Real;
      HBL_TT_24 : Real;
      HBL_TT_25 : Real;
      HBL_TT_26 : Real;
      HBL_TT_27 : Real;
      CPC_CT_851 : Real;
      CPC_HCV_853_A1 : Real;
      CPC_PT_862 : Real;
      CPC_PT_865 : Real;
      CPC_TT_866 : Real;
      CPC_TT_871 : Real;
      CPC_PT_872 : Real;
      CPC_HCV_880_A1 : Real;
      HBL_HCV_900_A1 : Real;
      HBL_TT_901 : Real;
      HBL_PT_902 : Real;
      HBL_FT_903 : Real;
      HBL_CT_950 : Real;
      HBL_CT_951 : Real;
      HBL_PT_960 : Real;
      HBL_PT_961 : Real;
      CompressorVolumetricEfficiency : Real;
      CompressorIsentropicEfficiency : Real;
      CompressorMassFlow : Real;
      HeatSinkPinch : Real;
      HeatSinkMassFlow : Real;
      HeatSourceHeatRate : Real;
      HeatSourcePinch : Real;
      HeatSourceMassFlow : Real;
   END_VAR
BEGIN
END_DATA_BLOCK

DATA_BLOCK "DB_ToHB"   // DB101
{ S7_Optimized_Access := 'FALSE' }
VERSION : 0.1
// stored: AutoNumber false, DBAccessibleFromOPCUA true, IsOnlyStoredInLoadMemory false, IsWriteProtectedInAS false
   VAR
      StartRequest : Bool;   // 1 = start Heatbooster, 0 = do nothing (level)
      StopRequest : Bool;   // 1 = stop, 0 = do nothing (overrides start signal) (level) (Regular stop, with cooldown periods etc)
      FastStopRequest : Bool;   // 1 = fast stop, 0 = do nothing (overrides start and stop signals) (level) (Stop NOW, but not Emergency Stop)
      EnableHeatbooster : Bool;   // 1 = allow operation, 0 = disable operation (level)
      AlarmAcknowledge : Bool;   // 1 = clear all alarms, 0 = do nothing (edge)
      ResetEmergencyStop : Bool;   // 1 = reset emergency stop, 0 = do nothing (edge)
      SpareCmd006 : Bool;   // 1 = Ventilation ok, 0 = ignore start command
      SpareCmd007 : Bool;   // 1 = Detected (stop request), 0 = do nothing
      SpareCmd010 : Bool;
      SpareCmd011 : Bool;
      SpareCmd012 : Bool;
      SpareCmd013 : Bool;
      SpareCmd014 : Bool;
      SpareCmd015 : Bool;
      SpareCmd016 : Bool;
      SpareCmd017 : Bool;
      WatchdogCounter : UInt;   // Liveness counter (free-running)
      Setpoint : Real;   // [%] Heatbooster setpoint
      SpareStatus080 : Bool;
      SpareStatus081 : Bool;
      SpareStatus082 : Bool;
      SpareStatus083 : Bool;
      SpareStatus084 : Bool;
      SpareStatus085 : Bool;
      SpareStatus086 : Bool;
      SpareStatus087 : Bool;
      SpareStatus090 : Bool;
      SpareStatus091 : Bool;
      SpareStatus092 : Bool;
      SpareStatus093 : Bool;
      SpareStatus094 : Bool;
      SpareStatus095 : Bool;
      SpareStatus096 : Bool;
      SpareStatus097 : Bool;
      Spare10 : Real;
      Spare14 : Real;
      Spare18 : Real;
      Spare22 : Real;
      Spare26 : Real;
      Spare30 : Real;
      Spare34 : Real;
      Spare38 : Real;
      ProteinDryerTemperature : Real;
      StarchDryerTemperature : Real;
      HBhallRelativeHumidity : Real;
      HBhallGasDetector : Real;
      StarchDryerAirInTemperature : Real;
      StarchDryerAirOutTemperature : Real;
      ProteinDryerAirInTemperature : Real;
      ProteinDryerAirOutTemperature : Real;
   END_VAR
BEGIN
END_DATA_BLOCK

DATA_BLOCK "CAN_Data_DB"   // DB3
{ S7_Optimized_Access := 'TRUE' }
VERSION : 0.1
// stored: AutoNumber true, DBAccessibleFromOPCUA true, IsOnlyStoredInLoadMemory false, IsRetainMemResEnabled false, IsWriteProtectedInAS false, MemoryReserve 100
   VAR
      InputData : Struct   // Receive
         CAN_ID_101h : Struct
            StartRequest : Bool;
            StopRequest : Bool;
            Clearance : Bool;
            PumaSystemReady : Bool;
            AlarmAcknowledge : Bool;
            ResetEmergencyStop : Bool;
            FastStopRequest : Bool;
            HydrolockProtection : Bool;
            ForceSuperheatSP : Bool;
            ForceHeatSinkOutSP : Bool;
            ForcePerformanceControlSP : Bool;
            ForceOilHeatingSP : Bool;
            ForceExpansionValveSP : Bool;
            ForcePinchSP : Bool;
            SpareByte2Bit6 : Bool;
            SpareByte2Bit7 : Bool;
            WatchdogFeedback : Word;
            I_326 : Bool;   // 0
            I_327 : Bool;   // 1
            I_330 : Bool;   // 2
            I_372 : Bool;   // 3
            I_373 : Bool;   // 4
            Spare55 : Bool;   // 5
            Spare56 : Bool;   // 6
            Spare57 : Bool;   // 7
            Spare60 : Bool;   // 0
            Spare61 : Bool;   // 1
            Spare62 : Bool;   // 2
            Spare63 : Bool;   // 3
            Spare64 : Bool;   // 4
            Spare65 : Bool;   // 5
            Spare66 : Bool;   // 6
            Spare67 : Bool;   // 7
            SpareByte7 : Byte;
            SpareByte8 : Byte;
         END_STRUCT;
         CAN_ID_102h : Struct
            SuperheatSP : Real;
            HeatSinkOutSP : Real;
         END_STRUCT;
         CAN_ID_103h : Struct
            PerformanceControlSP : Real;
            OilHeatingSP : Real;
         END_STRUCT;
         CAN_ID_104h : Struct
            ExpansionValveSP : Real;
            PinchSP : Real;
         END_STRUCT;
         CAN_ID_105h : Struct
            ThermalPowerOutput : Real;
            ThermalPowerInput : Real;
         END_STRUCT;
         CAN_ID_110h : Struct
            I_208 : Real;
            I_209 : Real;
         END_STRUCT;
         CAN_ID_111h : Struct
            I_210 : Real;
            I_211 : Real;
         END_STRUCT;
         CAN_ID_112h : Struct
            I_206 : Real;
            E_214 : Real;
         END_STRUCT;
         CAN_ID_113h : Struct
            I_302 : Real;
            E_213 : Real;
         END_STRUCT;
         CAN_ID_114h : Struct
            I_301 : Real;
            I_201 : Real;
         END_STRUCT;
         CAN_ID_115h : Struct
            I_202 : Real;
            I_307 : Real;
         END_STRUCT;
         CAN_ID_116h : Struct
            I_355 : Real;
            I_308 : Real;
         END_STRUCT;
         CAN_ID_117h : Struct
            I_300 : Real;
            I_301 : Real;
         END_STRUCT;
         CAN_ID_118h : Struct
            I_304 : Real;
            I_306 : Real;
         END_STRUCT;
         CAN_ID_119h : Struct
            I_320 : Real;
            I_321 : Real;
         END_STRUCT;
         CAN_ID_120h : Struct
            I_322 : Real;
            I_323 : Real;
         END_STRUCT;
         CAN_ID_121h : Struct
            I_324 : Real;
            I_328 : Real;
         END_STRUCT;
         CAN_ID_122h : Struct
            I_350 : Real;
            I_351 : Real;
         END_STRUCT;
         CAN_ID_123h : Struct
            I_354 : Real;
            I_356 : Real;
         END_STRUCT;
         CAN_ID_124h : Struct
            I_370 : Real;
            I_374 : Real;
         END_STRUCT;
         CAN_ID_125h : Struct
            E_301 : Real;
            E_330 : Real;
         END_STRUCT;
         CAN_ID_126h : Struct
            E_351 : Real;
            Spare : Real;
         END_STRUCT;
      END_STRUCT;
      OutputData { S7_SetPoint := 'True'} : "CAN-IDs_ToSend";   // Send
   END_VAR
BEGIN
   OutputData.IDs[5] := 16#0210;
   OutputData.IDs[6] := 16#0211;
   OutputData.IDs[7] := 16#0212;
   OutputData.IDs[8] := 16#0213;
   OutputData.IDs[9] := 16#0214;
   OutputData.IDs[10] := 16#0215;
   OutputData.IDs[11] := 16#0216;
   OutputData.IDs[12] := 16#0217;
   OutputData.IDs[13] := 16#0218;
   OutputData.IDs[14] := 16#0219;
   OutputData.IDs[15] := 16#0220;
   OutputData.IDs[16] := 16#0221;
   OutputData.IDs[17] := 16#0222;
   OutputData.IDs[18] := 16#0223;
   OutputData.IDs[19] := 16#0224;
   OutputData.IDs[20] := 16#0225;
   OutputData.IDs[21] := 16#0226;
   OutputData.IDs[22] := 16#0227;
   OutputData.IDs[23] := 16#0228;
   OutputData.IDs[24] := 16#0229;
   OutputData.IDs[25] := 16#0231;
   OutputData.IDs[26] := 16#0232;
   OutputData.IDs[27] := 16#0235;
   OutputData.IDs[28] := 16#0236;
   OutputData.IDs[29] := 16#0237;
   OutputData.IDs[30] := 16#0238;
   OutputData.IDs[31] := 16#0239;
   OutputData.IDs[32] := 16#0240;
   OutputData.IDs[33] := 16#0241;
   OutputData.IDs[34] := 16#0242;
   OutputData.IDs[35] := 16#0243;
   OutputData.IDs[36] := 16#0244;
   OutputData.IDs[37] := 16#0245;
   OutputData.IDs[38] := 16#0246;
   OutputData.IDs[39] := 16#0247;
   OutputData.IDs[40] := 16#0248;
   OutputData.IDs[41] := 16#0250;
   OutputData.IDs[42] := 16#0251;
   OutputData.IDs[43] := 16#0252;
   OutputData.IDs[44] := 16#0253;
   OutputData.IDs[45] := 16#0254;
   OutputData.IDs[46] := 16#0255;
   OutputData.IDs[47] := 16#0256;
   OutputData.IDs[48] := 16#0257;
   OutputData.IDs[49] := 16#0258;
   OutputData.IDs[50] := 16#0259;
   OutputData.IDs[51] := 16#0260;
   OutputData.IDs[52] := 16#0261;
   OutputData.IDs[53] := 16#0262;
   OutputData.IDs[54] := 16#0263;
   OutputData.IDs[55] := 16#0264;
   OutputData.IDs[56] := 16#0265;
   OutputData.IDs[57] := 16#0266;
   OutputData.IDs[58] := 16#0301;
   OutputData.IDs[59] := 16#0302;
   OutputData.IDs[60] := 16#0303;
   OutputData.IDs[61] := 16#0304;
   OutputData.IDs[62] := 16#0311;
   OutputData.IDs[63] := 16#0312;
   OutputData.IDs[64] := 16#0313;
   OutputData.IDs[65] := 16#0314;
   OutputData.IDs[66] := 16#0315;
   OutputData.IDs[67] := 16#0305;
   OutputData.IDs[68] := 16#0230;
END_DATA_BLOCK

DATA_BLOCK "DB_Puma"   // DB7
{ S7_Optimized_Access := 'TRUE' }
VERSION : 0.1
// stored: AutoNumber true, DBAccessibleFromOPCUA true, IsOnlyStoredInLoadMemory false, IsRetainMemResEnabled false, IsWriteProtectedInAS false, MemoryReserve 100
   VAR
      Watchdog : "stHeartbeatCount2";   // Comm monitoring Puma <-> Heatbooster
      "CAN-Reset_Required" { S7_SetPoint := 'True'} : Bool;   // Manually reset the CAN comm
   END_VAR
BEGIN
   Watchdog.bEnable := true;
   Watchdog.tTimeout := T#2s;
END_DATA_BLOCK

DATA_BLOCK "MasterData"   // DB13
{ S7_Optimized_Access := 'FALSE' }
VERSION : 0.1
// stored: AutoNumber true, DBAccessibleFromOPCUA true, IsOnlyStoredInLoadMemory false, IsWriteProtectedInAS false
   VAR
      dataPtr : "typeDataPtr";
   END_VAR
BEGIN
END_DATA_BLOCK

DATA_BLOCK "DB_Application"   // DB9
{ S7_Optimized_Access := 'FALSE' }
VERSION : 0.1
// stored: AutoNumber true, DBAccessibleFromOPCUA true, IsOnlyStoredInLoadMemory false, IsWriteProtectedInAS false
   VAR
      ToHB : Struct
         StartRequest : Bool;
         StopRequest : Bool;
         AlarmAcknowledge : Bool;
         EmergencyStopResetRequest : Bool;
         FastStopRequest : Bool;
         HydrolockProtection : Bool;
         SpareCommand6 : Bool;
         SpareCommand7 : Bool;
         SuperheatManualMode : Bool;
         HeatSinkOutManualMode : Bool;
         PerformanceControlManualMode : Bool;
         OilHeatingRegulatorManualMode : Bool;
         ExpansionValveRegulatorManualMode : Bool;
         PinchRegulatorManualMode : Bool;
         SpareManualMode6 : Bool;
         SpareManualMode7 : Bool;
         PumaCommOk : Bool;   // 1 = communication OK, 0 = communication dead
         HeatSourceOk : Bool;   // 1 = Source ready, 0 = source not ready
         HeatSinkOk : Bool;   // 1 = Sink ready, 0 = sink not ready
         SpareGroup2Command3 : Bool;
         SpareGroup2Command4 : Bool;
         SpareGroup2Command5 : Bool;
         SpareGroup2Command6 : Bool;
         SpareGroup2Command7 : Bool;
         SpareGroup3Command0 : Bool;
         SpareGroup3Command1 : Bool;
         SpareGroup3Command2 : Bool;
         SpareGroup3Command3 : Bool;
         SpareGroup3Command4 : Bool;
         SpareGroup3Command5 : Bool;
         SpareGroup3Command6 : Bool;
         SpareGroup3Command7 : Bool;
         SuperheatManualValue : Real;
         HeatSinkOutManualValue : Real;
         PerformanceControlManualValue : Real;
         OilHeatingManualValue : Real;
         ExpansionValveManualValue : Real;
         PinchManualValue : Real;
         HeatboosterSetpoint : Real;
         RegulationTarget : Int;
         LivenessCounter : UInt;
         HBL_HCV_514_A1 : Real;   // If externally controlled
         HBL_HCV_548_A1 : Real;   // If externally controlled
         HBL_TT_546 : Real;   // If externally controlled
         HBL_PT_547 : Real;   // If externally controlled
         HBL_HCV_515_A1 : Real;   // If externally controlled
         HBL_TT_901 : Real;   // If externally controlled
         HBL_PT_902 : Real;   // If externally controlled
         HBL_TT_512 : Real;   // If externally controlled
         HBL_PT_511 : Real;   // If externally controlled
         HBL_PT_519 : Real;   // If externally controlled
         HBL_TT_518 : Real;   // If externally controlled
      END_STRUCT;
      FromHB : Struct
         EmergencyStop : Bool;
         OilHeatersGroup1 : Bool;
         OilHeatersGroup2 : Bool;
         HBL_SC_01_Ready : Bool;
         HBL_SC_01_Run : Bool;
         HBL_SC_01_Tripped : Bool;
         HBL_SC_02_Ready : Bool;
         HBL_SC_02_Run : Bool;
         HBL_SC_02_Tripped : Bool;
         HBL_SC_10_Ready : Bool;
         HBL_SC_10_Run : Bool;
         HBL_SC_10_Tripped : Bool;
         HBL_HV_630 : Bool;
         HBL_HV_631 : Bool;
         HBL_HV_860 : Bool;
         HBL_HV_861 : Bool;
         HBL_HV_114 : Bool;
         HBL_HV_115 : Bool;
         CPC_P_01 : Bool;
         SSC_P_01 : Bool;
         SSC_F_01 : Bool;
         SSC_P_02 : Bool;
         HBL_LS_01 : Bool;
         HBL_LS_02 : Bool;
         HBL_HV_112 : Bool;
         HBL_HV_113 : Bool;
         HBL_LSH_62 : Bool;
         HBL_LSL_63 : Bool;
         HBL_LSH_64 : Bool;
         HBL_LSL_864 : Bool;
         HBL_LS_632 : Bool;
         HBL_LS_633 : Bool;
         HBL_SC_03_Ready : Bool;
         HBL_SC_03_Run : Bool;
         HBL_SC_03_Tripped : Bool;
         HBL_HCV_514_Force : Bool;
         HBL_HCV_548_Force : Bool;
         Spare05 : Bool;
         Spare06 : Bool;
         Spare07 : Bool;
         MachineState : Int;
         CompressorType : Int;
         SystemType : Int;
         RefrigerantType : Int;
         UptimeHours : Int;
         UptimeMinutes : Int;
         UptimeSeconds : Int;
         ActiveTimeHours : Int;
         ActiveTimeMinutes : Int;
         ActiveTimeSeconds : Int;
         RunningTimeHours : Int;
         RunningTimeMinutes : Int;
         RunningTimeSeconds : Int;
         Alarms : Array[0..191] of Bool;   // Compressed alarm bits
         HeatboosterSetpoint : Real;
         RegulationTarget : Int;
         HBL_HCV_514 : Real;   // Force setpoint
         HBL_HCV_548 : Real;   // Force setpoint
         DB_AI : Struct
            HBL_TT_502 : Real;
            HBL_PT_503 : Real;
            HBL_TT_504 : Real;
            HBL_LT_510 : Real;
            HBL_PT_511 : Real;
            HBL_TT_512 : Real;
            HBL_TT_516 : Real;
            HBL_PT_517 : Real;
            HBL_TT_518 : Real;
            HBL_PT_519 : Real;
            HBL_FT_520 : Real;
            HBL_TT_530 : Real;
            HBL_PT_531 : Real;
            HBL_TT_532 : Real;
            HBL_TT_533 : Real;
            HBL_PT_534 : Real;
            HBL_AT_535 : Real;
            HBL_TT_540 : Real;
            HBL_PT_541 : Real;
            HBL_TT_542 : Real;
            HBL_TT_543 : Real;
            HBL_PT_544 : Real;
            HBL_AT_545 : Real;
            HBL_TT_546 : Real;
            HBL_PT_547 : Real;
            HBL_TT_571 : Real;
            HBL_PT_572 : Real;
            HBL_TT_573 : Real;
            HBL_LT_610 : Real;
            HBL_TT_611 : Real;
            HBL_PT_612 : Real;
            HBL_CT_615 : Real;
            HBL_PT_618 : Real;
            HBL_PT_635 : Real;
            HBL_PT_636 : Real;
            HBL_LT_650 : Real;
            HBL_PT_651 : Real;
            HBL_PT_701 : Real;
            HBL_PT_702 : Real;
            HBL_PT_703 : Real;
            CPC_LT_870 : Real;
            CPC_TT_871 : Real;
            CPC_PT_872 : Real;
            CPC_PT_862 : Real;
            HBL_TT_901 : Real;
            HBL_PT_902 : Real;
            HBL_TT_03 : Real;
            HBL_TT_16 : Real;
            HBL_TT_17 : Real;
            HBL_TT_18 : Real;
            HBL_TT_20 : Real;
            HBL_TT_21 : Real;
            HBL_TT_22 : Real;
            HBL_TT_23 : Real;
            HBL_TT_24 : Real;
            HBL_TT_25 : Real;
            HBL_TT_26 : Real;
            HBL_TT_27 : Real;
            HBL_PT_05 : Real;
            HBL_PT_06 : Real;
            HBL_PT_17 : Real;
            HBL_CT_01 : Real;
            HBL_CT_03 : Real;
            SSC_TT_01 : Real;
            SSC_TT_02 : Real;
            SSC_TT_03 : Real;
            SSC_TT_04 : Real;
            SSC_PIT_01 : Real;
            SSC_PDT_01 : Real;
            SSC_LT_01 : Real;
         END_STRUCT;
         DB_Calc : Struct
            Compressor_CrankcaseSaturationTemperature : Real;
            Compressor_CrankcaseSuperheat : Real;
            Compressor_VolumetricEfficiency : Real;
            Compressor_IsentropicEfficiency : Real;
            Compressor_Massflow : Real;
            Heatsink_DeltaT : Real;
            Heatsink_Pinch : Real;
            Heatsink_Heatrate : Real;
            Heatsink_DeltaP : Real;
            Heatsink_Massflow : Real;
            Heatsource_DeltaT : Real;
            Heatsource_Pinch : Real;
            Heatsource_Heatrate : Real;
            Heatsource_DeltaP : Real;
            Heatsource_TemperatureRateOfChange : Real;
            Heatsource_Massflow : Real;
            HighPressPart_CompressorSaturationTemperature : Real;
            HighPressPart_CompressorSuperheat : Real;
            HighPressPart_CondenserSaturationTemperature : Real;
            HighPressPart_CondenserSubcooling : Real;
            HighPressPart_ExpansionValveSubcooling : Real;
            HighPressPart_CondenserDeltaP : Real;
            LowPressPart_EvaporatorSuperheat : Real;
            LowPressPart_CompressorSuperheat : Real;
            LowPressPart_EvaporatorSaturationTemperature : Real;
            LowPressPart_CompressorSaturationTemperature : Real;
            System_Quality : Real;
            System_COP : Real;
            System_ElectricalPower : Real;
            System_TemperatureLift : Real;
            System_MotorEfficiency : Real;
            System_FMEP : Real;
            Aux_ShaftSealDeltaT : Real;
            Aux_CPCPumpDeltaP : Real;
            Misc_EvaporatorDischargePressureMean : Real;
            Misc_EvaporatorDischargeTemperatureMin : Real;
            Misc_EvaporatorDischargeTemperatureMean : Real;
            Misc_OilFilterDeltaP : Real;
         END_STRUCT;
         DB_InverterDrives : Struct
            HBL_SC_01_A1 : Real;
            HBL_SC_01_A2 : Real;
            HBL_SC_01_A3 : Real;
            HBL_SC_02_A1 : Real;
            HBL_SC_02_A2 : Real;
            HBL_SC_02_A3 : Real;
            HBL_SC_10_A1 : Real;
            HBL_SC_10_A2 : Real;
            HBL_SC_10_A3 : Real;
            HBL_SC_03_A1 : Real;
            HBL_SC_03_A2 : Real;
            HBL_SC_03_A3 : Real;
         END_STRUCT;
         DB_Valves : Struct
            HBL_HCV_576_A1 : Real;
            HBL_HCV_578_A1 : Real;
            HBL_HCV_577_A1 : Real;
            HBL_HCV_579_A1 : Real;
            HBL_HCV_515_A1 : Real;
            HBL_HCV_575_A1 : Real;
            HBL_HCV_616_A1 : Real;
            HBL_HCV_700_A1 : Real;
            HBL_HCV_514_A1 : Real;
            HBL_HCV_548_A1 : Real;
         END_STRUCT;
      END_STRUCT;
   END_VAR
BEGIN
END_DATA_BLOCK

ORGANIZATION_BLOCK "Main"   // OB1, FBD, ProgramCycle
TITLE = "Main Program Sweep (Cycle)"
{ S7_Optimized_Access := 'TRUE' }
VERSION : 0.1
// stored: AutoNumber true, IsIECCheckEnabled false, SetENOAutomatically false
   VAR_INPUT
      Initial_Call : Bool;
      Remanence : Bool;
   END_VAR
BEGIN

REGION Network 1: Land on Mars
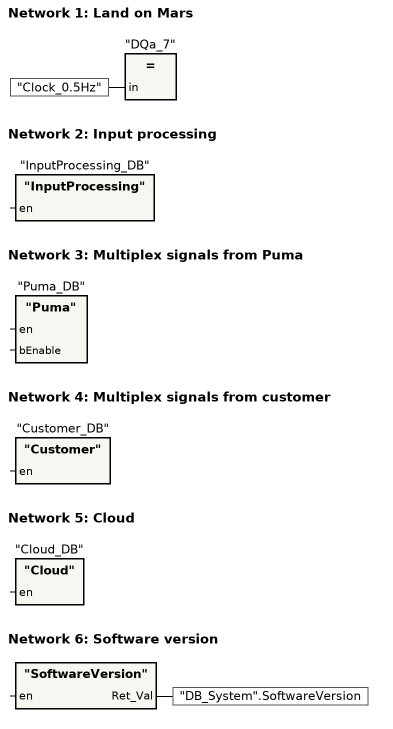
   "DQa_7" := "Clock_0.5Hz";
END_REGION

REGION Network 2: Input processing
   "InputProcessing_DB"();   // "InputProcessing"
END_REGION

REGION Network 3: Multiplex signals from Puma
   "Puma_DB"();   // "Puma"
END_REGION

REGION Network 4: Multiplex signals from customer
   "Customer_DB"();   // "Customer"
END_REGION

REGION Network 5: Cloud
   "Cloud_DB"();   // "Cloud"
END_REGION

REGION Network 6: Software version
   "DB_System".SoftwareVersion := "SoftwareVersion"();
END_REGION
END_ORGANIZATION_BLOCK

FUNCTION_BLOCK "InputProcessing"   // FB48, FBD
{ S7_Optimized_Access := 'TRUE' }
AUTHOR : Heaten
VERSION : 0.1
// stored: AutoNumber false, IsIECCheckEnabled false, IsRetainMemResEnabled false, MemoryReserve 0, SetENOAutomatically false, UDAEnableTagReadback false
   VAR
      PumaInputProcessing : "PumaInputProcessing";
      CustomerInputProcessing { S7_SetPoint := 'True'} : "CustomerInputProcessing";
   END_VAR
BEGIN

REGION Network 1: Values from Puma
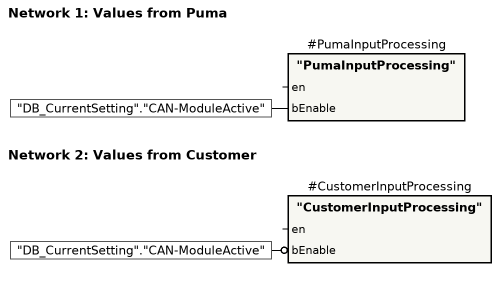
   #PumaInputProcessing(bEnable := "DB_CurrentSetting"."CAN-ModuleActive");   // "PumaInputProcessing"
END_REGION

REGION Network 2: Values from Customer
   #CustomerInputProcessing(bEnable := NOT "DB_CurrentSetting"."CAN-ModuleActive");   // "CustomerInputProcessing"
END_REGION

REGION Network 3: Analog inputs
   // Directly connected
END_REGION

REGION Network 4: Digital inputs
   // Directly connected
END_REGION
END_FUNCTION_BLOCK

FUNCTION_BLOCK "PumaInputProcessing"   // FB5, FBD
{ S7_Optimized_Access := 'TRUE' }
AUTHOR : Heaten
VERSION : 0.1
// stored: AutoNumber true, IsIECCheckEnabled false, IsRetainMemResEnabled false, MemoryReserve 0, SetENOAutomatically false, UDAEnableTagReadback false
   VAR_INPUT
      bEnable : Bool;
   END_VAR
   VAR
      Dummy : Bool;
   END_VAR
   VAR_TEMP
      bCommOk : Bool;   // Puma is running
      fDummy : Real;
   END_VAR
BEGIN

REGION Network 1: Comm ok
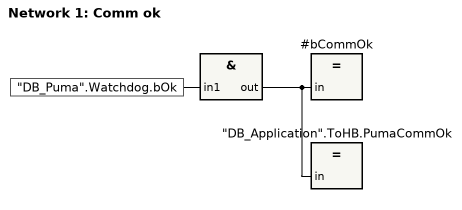
   #bCommOk := "DB_Puma".Watchdog.bOk;
   "DB_Application".ToHB.PumaCommOk := "DB_Puma".Watchdog.bOk;
END_REGION

REGION Network 2: Test Support System values (AI)
   // TSS = Test Support System
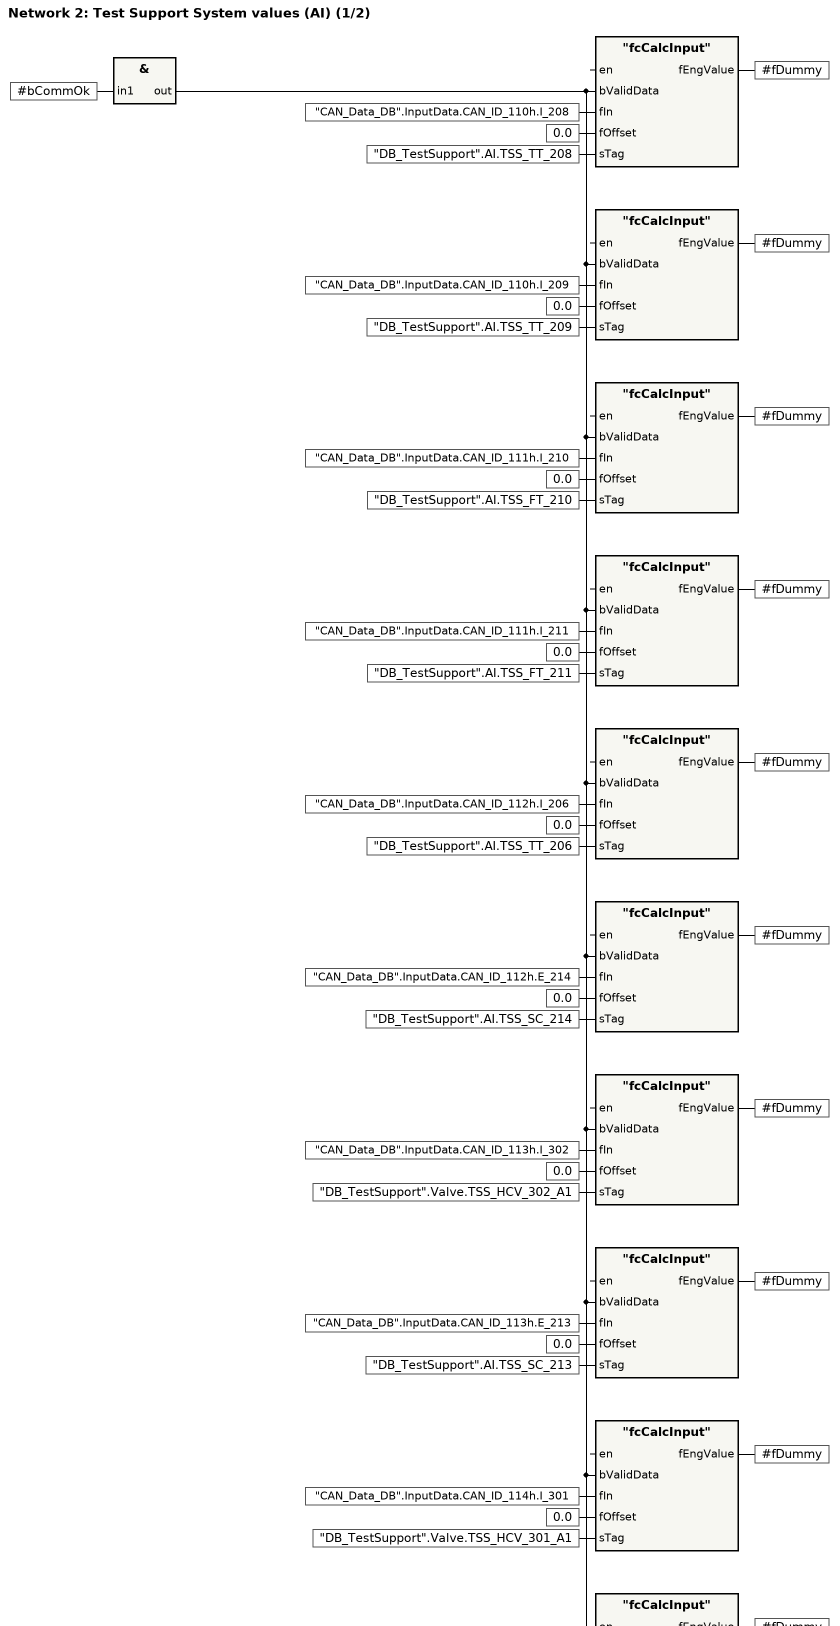
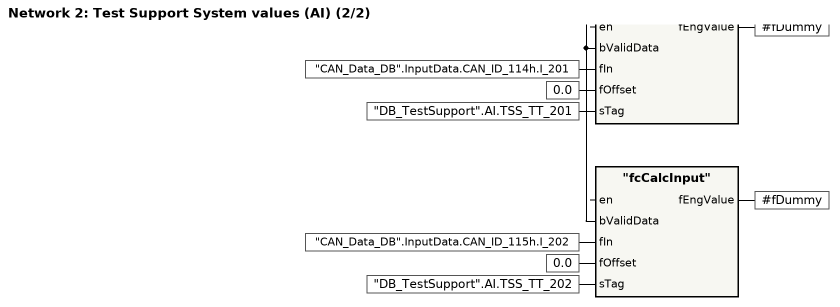
   "fcCalcInput"(bValidData := #bCommOk,
                 fIn := "CAN_Data_DB".InputData.CAN_ID_110h.I_208,
                 fOffset := 0.0,
                 sTag := "DB_TestSupport".AI.TSS_TT_208,
                 fEngValue => #fDummy);
   "fcCalcInput"(bValidData := #bCommOk,
                 fIn := "CAN_Data_DB".InputData.CAN_ID_110h.I_209,
                 fOffset := 0.0,
                 sTag := "DB_TestSupport".AI.TSS_TT_209,
                 fEngValue => #fDummy);
   "fcCalcInput"(bValidData := #bCommOk,
                 fIn := "CAN_Data_DB".InputData.CAN_ID_111h.I_210,
                 fOffset := 0.0,
                 sTag := "DB_TestSupport".AI.TSS_FT_210,
                 fEngValue => #fDummy);
   "fcCalcInput"(bValidData := #bCommOk,
                 fIn := "CAN_Data_DB".InputData.CAN_ID_111h.I_211,
                 fOffset := 0.0,
                 sTag := "DB_TestSupport".AI.TSS_FT_211,
                 fEngValue => #fDummy);
   "fcCalcInput"(bValidData := #bCommOk,
                 fIn := "CAN_Data_DB".InputData.CAN_ID_112h.I_206,
                 fOffset := 0.0,
                 sTag := "DB_TestSupport".AI.TSS_TT_206,
                 fEngValue => #fDummy);
   "fcCalcInput"(bValidData := #bCommOk,
                 fIn := "CAN_Data_DB".InputData.CAN_ID_112h.E_214,
                 fOffset := 0.0,
                 sTag := "DB_TestSupport".AI.TSS_SC_214,
                 fEngValue => #fDummy);
   "fcCalcInput"(bValidData := #bCommOk,
                 fIn := "CAN_Data_DB".InputData.CAN_ID_113h.I_302,
                 fOffset := 0.0,
                 sTag := "DB_TestSupport".Valve.TSS_HCV_302_A1,
                 fEngValue => #fDummy);
   "fcCalcInput"(bValidData := #bCommOk,
                 fIn := "CAN_Data_DB".InputData.CAN_ID_113h.E_213,
                 fOffset := 0.0,
                 sTag := "DB_TestSupport".AI.TSS_SC_213,
                 fEngValue => #fDummy);
   "fcCalcInput"(bValidData := #bCommOk,
                 fIn := "CAN_Data_DB".InputData.CAN_ID_114h.I_301,
                 fOffset := 0.0,
                 sTag := "DB_TestSupport".Valve.TSS_HCV_301_A1,
                 fEngValue => #fDummy);
   "fcCalcInput"(bValidData := #bCommOk,
                 fIn := "CAN_Data_DB".InputData.CAN_ID_114h.I_201,
                 fOffset := 0.0,
                 sTag := "DB_TestSupport".AI.TSS_TT_201,
                 fEngValue => #fDummy);
   "fcCalcInput"(bValidData := #bCommOk,
                 fIn := "CAN_Data_DB".InputData.CAN_ID_115h.I_202,
                 fOffset := 0.0,
                 sTag := "DB_TestSupport".AI.TSS_TT_202,
                 fEngValue => #fDummy);
END_REGION

REGION Network 3: Steam Adapter values (AI)
   // TSA = TSS Steam Adapters
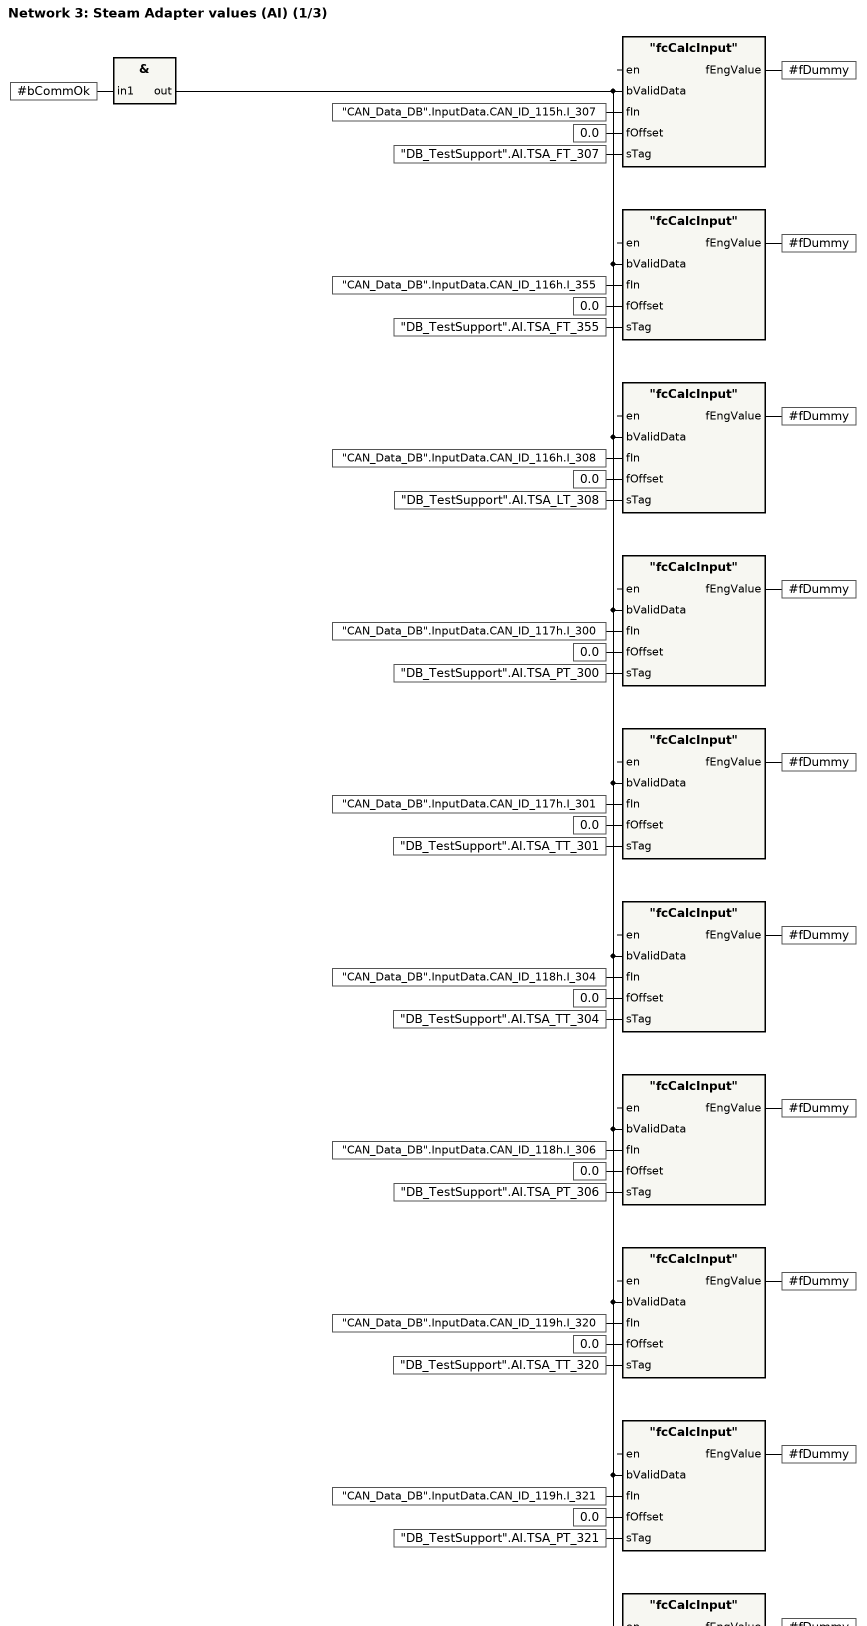
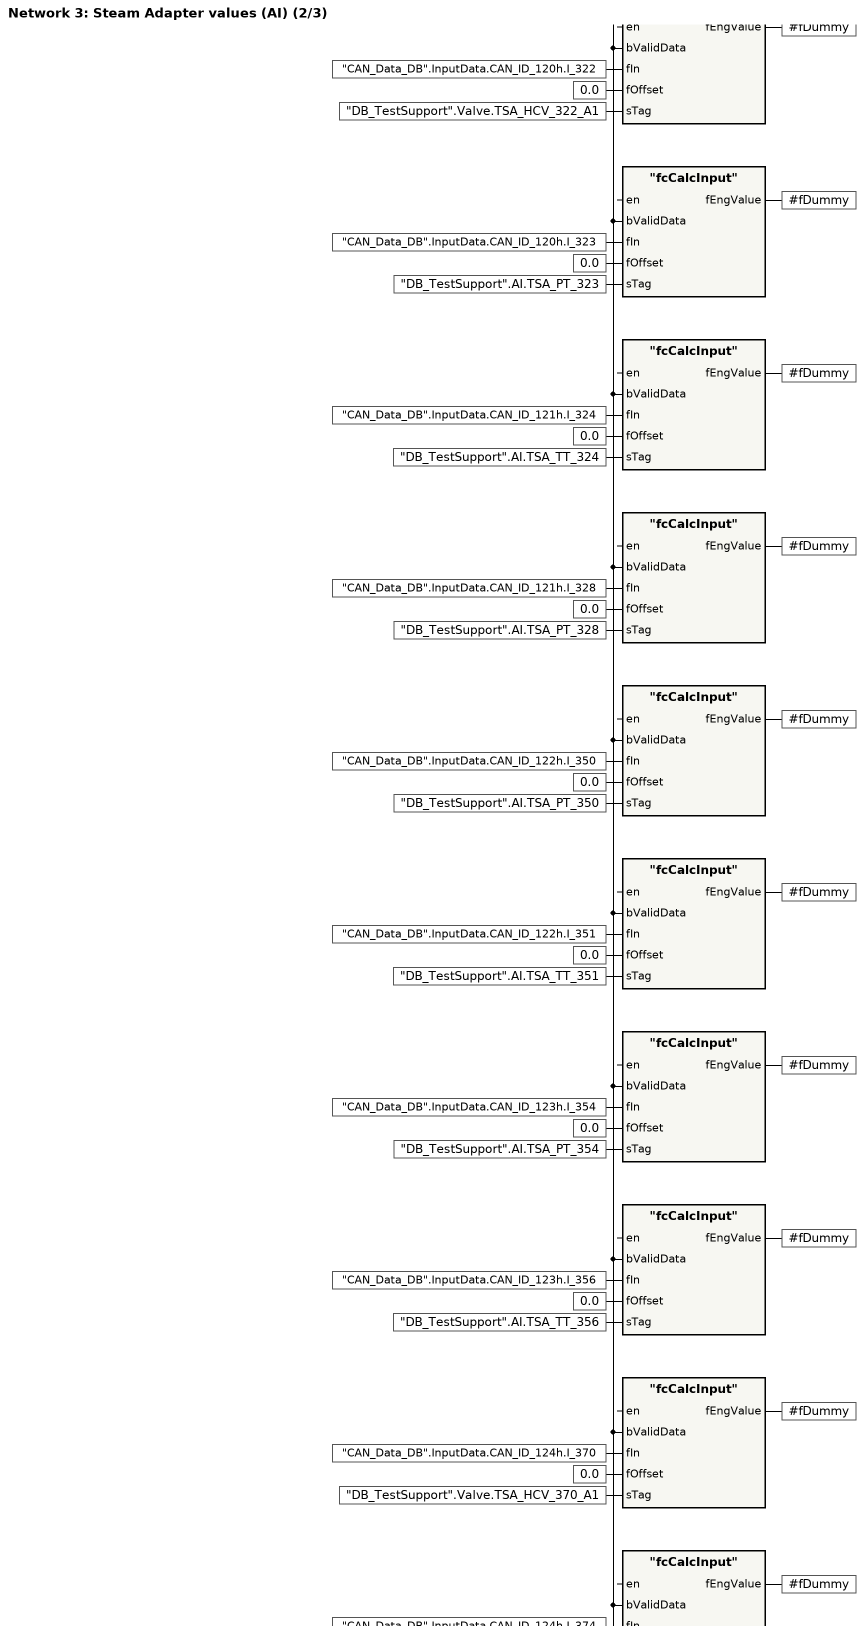
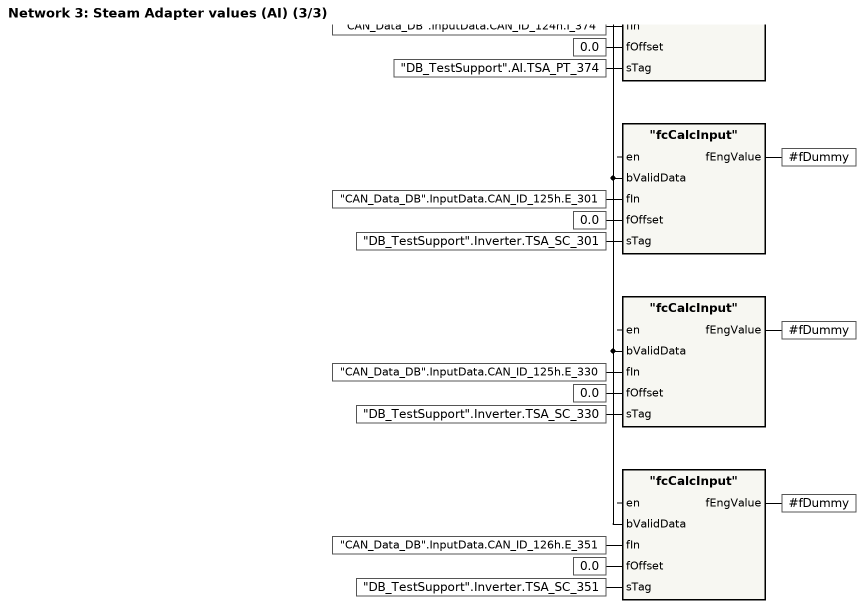
   "fcCalcInput"(bValidData := #bCommOk,
                 fIn := "CAN_Data_DB".InputData.CAN_ID_115h.I_307,
                 fOffset := 0.0,
                 sTag := "DB_TestSupport".AI.TSA_FT_307,
                 fEngValue => #fDummy);
   "fcCalcInput"(bValidData := #bCommOk,
                 fIn := "CAN_Data_DB".InputData.CAN_ID_116h.I_355,
                 fOffset := 0.0,
                 sTag := "DB_TestSupport".AI.TSA_FT_355,
                 fEngValue => #fDummy);
   "fcCalcInput"(bValidData := #bCommOk,
                 fIn := "CAN_Data_DB".InputData.CAN_ID_116h.I_308,
                 fOffset := 0.0,
                 sTag := "DB_TestSupport".AI.TSA_LT_308,
                 fEngValue => #fDummy);
   "fcCalcInput"(bValidData := #bCommOk,
                 fIn := "CAN_Data_DB".InputData.CAN_ID_117h.I_300,
                 fOffset := 0.0,
                 sTag := "DB_TestSupport".AI.TSA_PT_300,
                 fEngValue => #fDummy);
   "fcCalcInput"(bValidData := #bCommOk,
                 fIn := "CAN_Data_DB".InputData.CAN_ID_117h.I_301,
                 fOffset := 0.0,
                 sTag := "DB_TestSupport".AI.TSA_TT_301,
                 fEngValue => #fDummy);
   "fcCalcInput"(bValidData := #bCommOk,
                 fIn := "CAN_Data_DB".InputData.CAN_ID_118h.I_304,
                 fOffset := 0.0,
                 sTag := "DB_TestSupport".AI.TSA_TT_304,
                 fEngValue => #fDummy);
   "fcCalcInput"(bValidData := #bCommOk,
                 fIn := "CAN_Data_DB".InputData.CAN_ID_118h.I_306,
                 fOffset := 0.0,
                 sTag := "DB_TestSupport".AI.TSA_PT_306,
                 fEngValue => #fDummy);
   "fcCalcInput"(bValidData := #bCommOk,
                 fIn := "CAN_Data_DB".InputData.CAN_ID_119h.I_320,
                 fOffset := 0.0,
                 sTag := "DB_TestSupport".AI.TSA_TT_320,
                 fEngValue => #fDummy);
   "fcCalcInput"(bValidData := #bCommOk,
                 fIn := "CAN_Data_DB".InputData.CAN_ID_119h.I_321,
                 fOffset := 0.0,
                 sTag := "DB_TestSupport".AI.TSA_PT_321,
                 fEngValue => #fDummy);
   "fcCalcInput"(bValidData := #bCommOk,
                 fIn := "CAN_Data_DB".InputData.CAN_ID_120h.I_322,
                 fOffset := 0.0,
                 sTag := "DB_TestSupport".Valve.TSA_HCV_322_A1,
                 fEngValue => #fDummy);
   "fcCalcInput"(bValidData := #bCommOk,
                 fIn := "CAN_Data_DB".InputData.CAN_ID_120h.I_323,
                 fOffset := 0.0,
                 sTag := "DB_TestSupport".AI.TSA_PT_323,
                 fEngValue => #fDummy);
   "fcCalcInput"(bValidData := #bCommOk,
                 fIn := "CAN_Data_DB".InputData.CAN_ID_121h.I_324,
                 fOffset := 0.0,
                 sTag := "DB_TestSupport".AI.TSA_TT_324,
                 fEngValue => #fDummy);
   "fcCalcInput"(bValidData := #bCommOk,
                 fIn := "CAN_Data_DB".InputData.CAN_ID_121h.I_328,
                 fOffset := 0.0,
                 sTag := "DB_TestSupport".AI.TSA_PT_328,
                 fEngValue => #fDummy);
   "fcCalcInput"(bValidData := #bCommOk,
                 fIn := "CAN_Data_DB".InputData.CAN_ID_122h.I_350,
                 fOffset := 0.0,
                 sTag := "DB_TestSupport".AI.TSA_PT_350,
                 fEngValue => #fDummy);
   "fcCalcInput"(bValidData := #bCommOk,
                 fIn := "CAN_Data_DB".InputData.CAN_ID_122h.I_351,
                 fOffset := 0.0,
                 sTag := "DB_TestSupport".AI.TSA_TT_351,
                 fEngValue => #fDummy);
   "fcCalcInput"(bValidData := #bCommOk,
                 fIn := "CAN_Data_DB".InputData.CAN_ID_123h.I_354,
                 fOffset := 0.0,
                 sTag := "DB_TestSupport".AI.TSA_PT_354,
                 fEngValue => #fDummy);
   "fcCalcInput"(bValidData := #bCommOk,
                 fIn := "CAN_Data_DB".InputData.CAN_ID_123h.I_356,
                 fOffset := 0.0,
                 sTag := "DB_TestSupport".AI.TSA_TT_356,
                 fEngValue => #fDummy);
   "fcCalcInput"(bValidData := #bCommOk,
                 fIn := "CAN_Data_DB".InputData.CAN_ID_124h.I_370,
                 fOffset := 0.0,
                 sTag := "DB_TestSupport".Valve.TSA_HCV_370_A1,
                 fEngValue => #fDummy);
   "fcCalcInput"(bValidData := #bCommOk,
                 fIn := "CAN_Data_DB".InputData.CAN_ID_124h.I_374,
                 fOffset := 0.0,
                 sTag := "DB_TestSupport".AI.TSA_PT_374,
                 fEngValue => #fDummy);
   "fcCalcInput"(bValidData := #bCommOk,
                 fIn := "CAN_Data_DB".InputData.CAN_ID_125h.E_301,
                 fOffset := 0.0,
                 sTag := "DB_TestSupport".Inverter.TSA_SC_301,
                 fEngValue => #fDummy);
   "fcCalcInput"(bValidData := #bCommOk,
                 fIn := "CAN_Data_DB".InputData.CAN_ID_125h.E_330,
                 fOffset := 0.0,
                 sTag := "DB_TestSupport".Inverter.TSA_SC_330,
                 fEngValue => #fDummy);
   "fcCalcInput"(bValidData := #bCommOk,
                 fIn := "CAN_Data_DB".InputData.CAN_ID_126h.E_351,
                 fOffset := 0.0,
                 sTag := "DB_TestSupport".Inverter.TSA_SC_351,
                 fEngValue => #fDummy);
END_REGION

REGION Network 4: Steam Adapter values (DI)
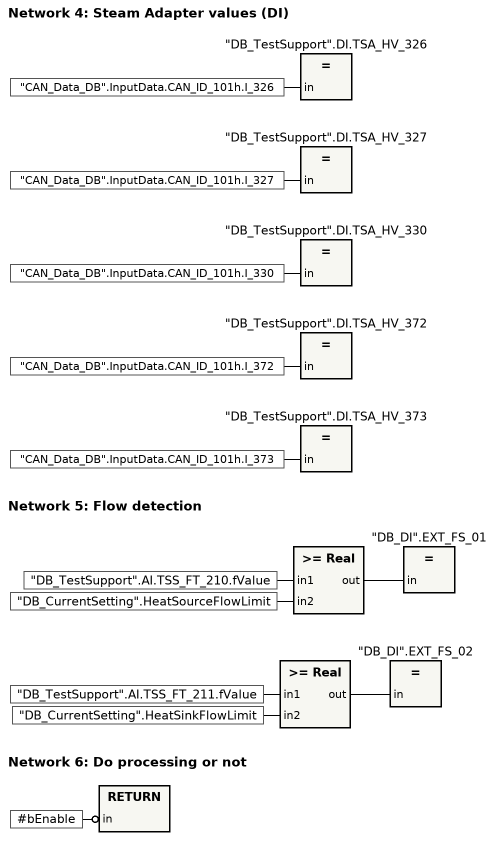
   "DB_TestSupport".DI.TSA_HV_326 := "CAN_Data_DB".InputData.CAN_ID_101h.I_326;
   "DB_TestSupport".DI.TSA_HV_327 := "CAN_Data_DB".InputData.CAN_ID_101h.I_327;
   "DB_TestSupport".DI.TSA_HV_330 := "CAN_Data_DB".InputData.CAN_ID_101h.I_330;
   "DB_TestSupport".DI.TSA_HV_372 := "CAN_Data_DB".InputData.CAN_ID_101h.I_372;
   "DB_TestSupport".DI.TSA_HV_373 := "CAN_Data_DB".InputData.CAN_ID_101h.I_373;
END_REGION

REGION Network 5: Flow detection
   "DB_DI".EXT_FS_01 := "DB_TestSupport".AI.TSS_FT_210.fValue >= "DB_CurrentSetting".HeatSourceFlowLimit;
   "DB_DI".EXT_FS_02 := "DB_TestSupport".AI.TSS_FT_211.fValue >= "DB_CurrentSetting".HeatSinkFlowLimit;
END_REGION

REGION Network 6: Do processing or not
   IF NOT #bEnable THEN
       ENO := TRUE;
       RETURN;
   END_IF;
END_REGION
END_FUNCTION_BLOCK

FUNCTION_BLOCK "CustomerInputProcessing"   // FB6, FBD
TITLE = Internalize customer values
{ S7_Optimized_Access := 'TRUE' }
AUTHOR : Heaten
VERSION : 0.1
// stored: AutoNumber true, IsIECCheckEnabled false, IsRetainMemResEnabled false, MemoryReserve 0, SetENOAutomatically false, UDAEnableTagReadback false
   VAR_INPUT
      bEnable : Bool;
   END_VAR
   VAR
      Dummy : Bool;
   END_VAR
BEGIN

REGION Network 1: Customer comm ok
END_REGION

REGION Network 2: Do processing or not
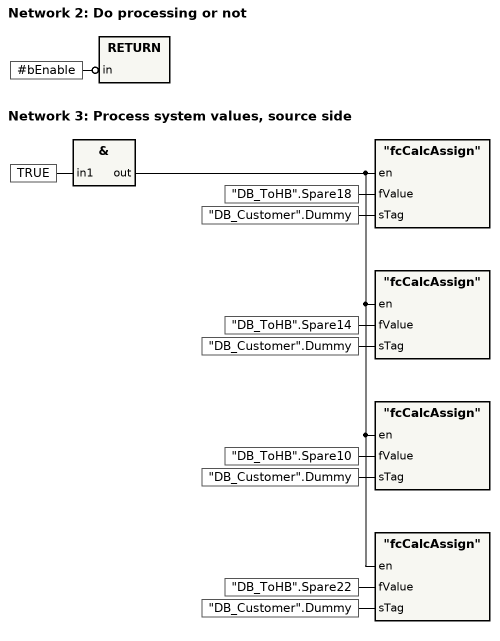
   IF NOT #bEnable THEN
       ENO := TRUE;
       RETURN;
   END_IF;
END_REGION

REGION Network 3: Process system values, source side
   IF TRUE THEN
       "fcCalcAssign"(fValue := "DB_ToHB".Spare18, sTag := "DB_Customer".Dummy);
       "fcCalcAssign"(fValue := "DB_ToHB".Spare14, sTag := "DB_Customer".Dummy);
       "fcCalcAssign"(fValue := "DB_ToHB".Spare10, sTag := "DB_Customer".Dummy);
       "fcCalcAssign"(fValue := "DB_ToHB".Spare22, sTag := "DB_Customer".Dummy);
   END_IF;
END_REGION

REGION Network 4: Beneo process system values, sink side
   // Including dryer air temperatures & Hall ambient measurements
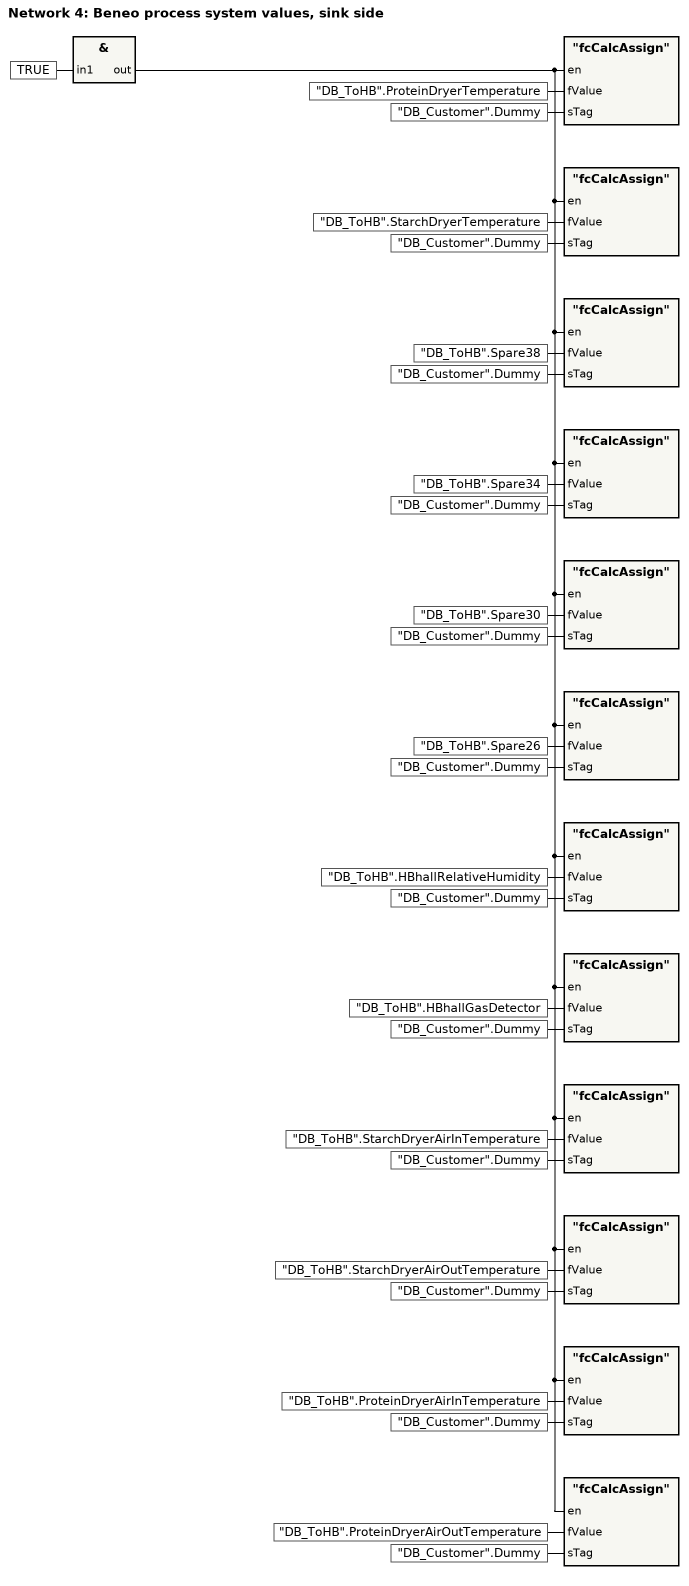
   IF TRUE THEN
       "fcCalcAssign"(fValue := "DB_ToHB".ProteinDryerTemperature, sTag := "DB_Customer".Dummy);
       "fcCalcAssign"(fValue := "DB_ToHB".StarchDryerTemperature, sTag := "DB_Customer".Dummy);
       "fcCalcAssign"(fValue := "DB_ToHB".Spare38, sTag := "DB_Customer".Dummy);
       "fcCalcAssign"(fValue := "DB_ToHB".Spare34, sTag := "DB_Customer".Dummy);
       "fcCalcAssign"(fValue := "DB_ToHB".Spare30, sTag := "DB_Customer".Dummy);
       "fcCalcAssign"(fValue := "DB_ToHB".Spare26, sTag := "DB_Customer".Dummy);
       "fcCalcAssign"(fValue := "DB_ToHB".HBhallRelativeHumidity, sTag := "DB_Customer".Dummy);
       "fcCalcAssign"(fValue := "DB_ToHB".HBhallGasDetector, sTag := "DB_Customer".Dummy);
       "fcCalcAssign"(fValue := "DB_ToHB".StarchDryerAirInTemperature, sTag := "DB_Customer".Dummy);
       "fcCalcAssign"(fValue := "DB_ToHB".StarchDryerAirOutTemperature, sTag := "DB_Customer".Dummy);
       "fcCalcAssign"(fValue := "DB_ToHB".ProteinDryerAirInTemperature, sTag := "DB_Customer".Dummy);
       "fcCalcAssign"(fValue := "DB_ToHB".ProteinDryerAirOutTemperature, sTag := "DB_Customer".Dummy);
   END_IF;
END_REGION

REGION Network 5: Flow detection
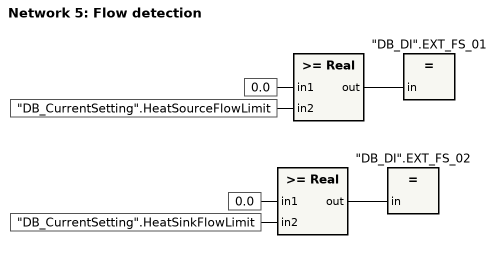
   "DB_DI".EXT_FS_01 := 0.0 >= "DB_CurrentSetting".HeatSourceFlowLimit;
   "DB_DI".EXT_FS_02 := 0.0 >= "DB_CurrentSetting".HeatSinkFlowLimit;
END_REGION
END_FUNCTION_BLOCK

FUNCTION_BLOCK "Puma"   // FB2, LAD
TITLE = Combine signals from Puma into DB_Application
{ S7_Optimized_Access := 'TRUE' }
VERSION : 0.1
// stored: AutoNumber true, IsIECCheckEnabled false, IsRetainMemResEnabled false, MemoryReserve 100, SetENOAutomatically false, UDAEnableTagReadback false
   VAR_INPUT
      bEnable : Bool;
   END_VAR
   VAR
      Watchdog : "fbHeartbeatCount2";
      Dummy { S7_SetPoint := 'True'} : UInt;
      epForceExpansionValveSP : Bool;
      enForceExpansionValveSP : Bool;
      epForceHeatSinkOutSP : Bool;
      enForceHeatSinkOutSP : Bool;
      epForceMotorRpmSP : Bool;
      enForceMotorRpmSP : Bool;
      epForceOilHeatingSP : Bool;
      enForceOilHeatingSP : Bool;
      epForcePinchSP : Bool;
      enForcePinchSP : Bool;
      epForceSuperheatSP : Bool;
      enForceSuperheatSP : Bool;
      epStartRequest : Bool;
      enStartRequest : Bool;
      epStopRequest : Bool;
      enStopRequest : Bool;
      epAlarmAcknowledge : Bool;
      enAlarmAcknowledge : Bool;
      epResetEmergencyStop : Bool;
      enResetEmergencyStop : Bool;
      epHydrolockProtection : Bool;
      enHydrolockProtection : Bool;
      enClearance : Bool;
      ExpansionManualPrev : Real;
      HeatSinkManualPrev : Real;
      PerformanceManualPrev : Real;
      OilHeatingManualPrev : Real;
      PinchManualPrev : Real;
      SuperheatManualPrev : Real;
      WatchdogTimeout : TON_TIME;
   END_VAR
   VAR_TEMP
      bStopReq : Bool;
      bWatchdogOk : Bool;
   END_VAR
   VAR_TEMP   // added for the SCL form of the ladder/FBD networks
      _w1 : Bool;
      _w2 : Bool;
      _w3 : Bool;
      _w4 : Bool;
      _w5 : Bool;
      _w6 : Bool;
      _w7 : Bool;
      _w8 : Bool;
      _w9 : Bool;
      _w10 : Bool;
      _w11 : Bool;
      _w12 : Bool;
   END_VAR
BEGIN

REGION Network 1: Watchdog
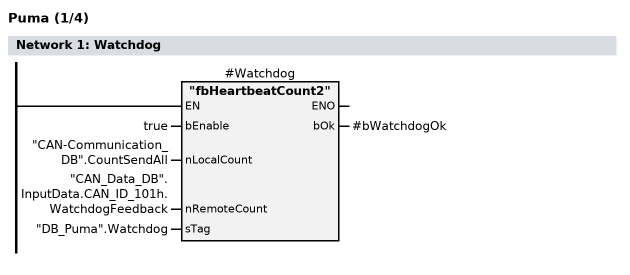
   RUNG wire#powerrail
      #Watchdog(bEnable := true, nLocalCount := "CAN-Communication_DB".CountSendAll, nRemoteCount := "CAN_Data_DB".InputData.CAN_ID_101h.WatchdogFeedback, sTag := "DB_Puma".Watchdog, bOk => #bWatchdogOk)
   END_RUNG
   // the same network as SCL:
   #Watchdog(bEnable := true,   // "fbHeartbeatCount2"
             nLocalCount := "CAN-Communication_DB".CountSendAll,
             nRemoteCount := "CAN_Data_DB".InputData.CAN_ID_101h.WatchdogFeedback,
             sTag := "DB_Puma".Watchdog,
             bOk => #bWatchdogOk);
END_REGION

REGION Network 2: Write Puma setpoints to Application
   // A positive edge followed by a SET  writes to the destination bit once, without "holding" the value. Easiest to write & read in ladder.
   // Triggering a MOVE on value change writes the value once without continually overwriting it.
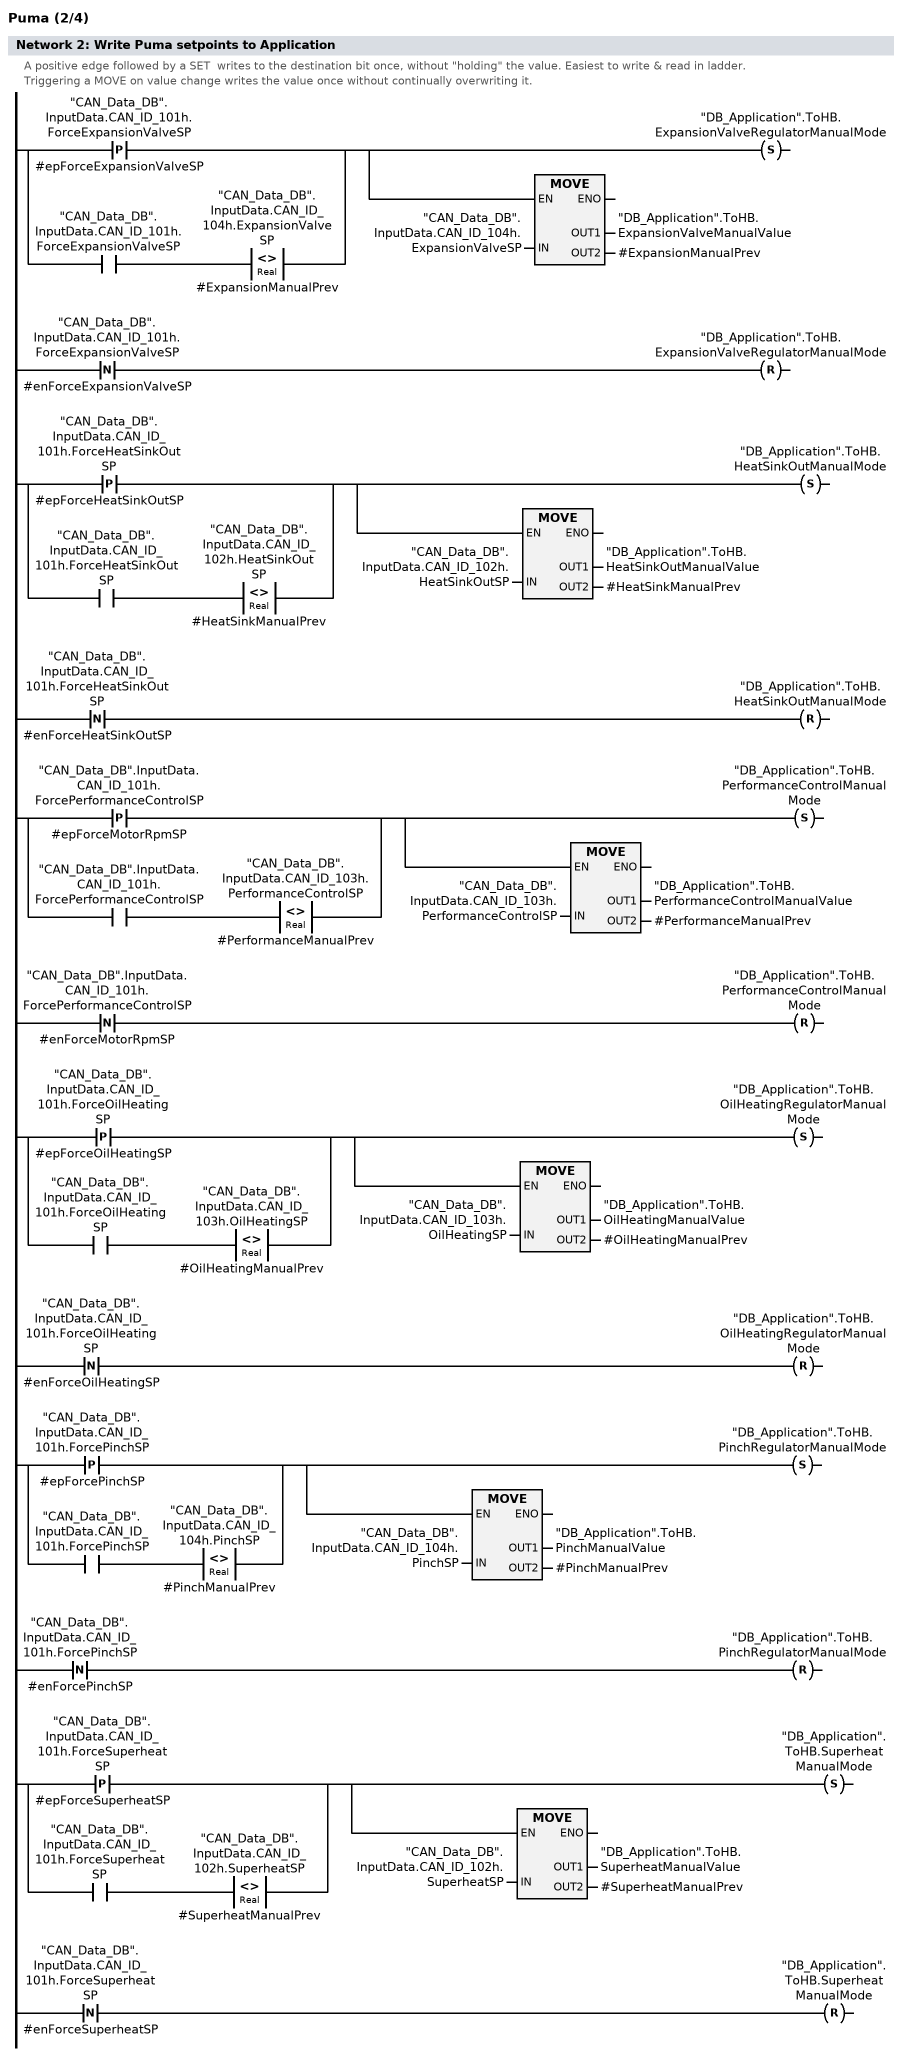
   RUNG wire#powerrail
      P_Contact(operand := "CAN_Data_DB".InputData.CAN_ID_101h.ForceExpansionValveSP, bit := #epForceExpansionValveSP)
      wire#w1
      S_Coil( "DB_Application".ToHB.ExpansionValveRegulatorManualMode )
   END_RUNG
   RUNG wire#powerrail
      Contact( "CAN_Data_DB".InputData.CAN_ID_101h.ForceExpansionValveSP )
      { S7_Templates := "SrcType := Real" } NE_Contact(in1 := "CAN_Data_DB".InputData.CAN_ID_104h.ExpansionValveSP, in2 := #ExpansionManualPrev)
   END_RUNG wire#w1
   RUNG wire#w1
      Move(in := "CAN_Data_DB".InputData.CAN_ID_104h.ExpansionValveSP, out1 => "DB_Application".ToHB.ExpansionValveManualValue, out2 => #ExpansionManualPrev)
   END_RUNG
   RUNG wire#powerrail
      N_Contact(operand := "CAN_Data_DB".InputData.CAN_ID_101h.ForceExpansionValveSP, bit := #enForceExpansionValveSP)
      R_Coil( "DB_Application".ToHB.ExpansionValveRegulatorManualMode )
   END_RUNG
   RUNG wire#powerrail
      P_Contact(operand := "CAN_Data_DB".InputData.CAN_ID_101h.ForceHeatSinkOutSP, bit := #epForceHeatSinkOutSP)
      wire#w2
      S_Coil( "DB_Application".ToHB.HeatSinkOutManualMode )
   END_RUNG
   RUNG wire#powerrail
      Contact( "CAN_Data_DB".InputData.CAN_ID_101h.ForceHeatSinkOutSP )
      { S7_Templates := "SrcType := Real" } NE_Contact(in1 := "CAN_Data_DB".InputData.CAN_ID_102h.HeatSinkOutSP, in2 := #HeatSinkManualPrev)
   END_RUNG wire#w2
   RUNG wire#w2
      Move(in := "CAN_Data_DB".InputData.CAN_ID_102h.HeatSinkOutSP, out1 => "DB_Application".ToHB.HeatSinkOutManualValue, out2 => #HeatSinkManualPrev)
   END_RUNG
   RUNG wire#powerrail
      N_Contact(operand := "CAN_Data_DB".InputData.CAN_ID_101h.ForceHeatSinkOutSP, bit := #enForceHeatSinkOutSP)
      R_Coil( "DB_Application".ToHB.HeatSinkOutManualMode )
   END_RUNG
   RUNG wire#powerrail
      P_Contact(operand := "CAN_Data_DB".InputData.CAN_ID_101h.ForcePerformanceControlSP, bit := #epForceMotorRpmSP)
      wire#w3
      S_Coil( "DB_Application".ToHB.PerformanceControlManualMode )
   END_RUNG
   RUNG wire#powerrail
      Contact( "CAN_Data_DB".InputData.CAN_ID_101h.ForcePerformanceControlSP )
      { S7_Templates := "SrcType := Real" } NE_Contact(in1 := "CAN_Data_DB".InputData.CAN_ID_103h.PerformanceControlSP, in2 := #PerformanceManualPrev)
   END_RUNG wire#w3
   RUNG wire#w3
      Move(in := "CAN_Data_DB".InputData.CAN_ID_103h.PerformanceControlSP, out1 => "DB_Application".ToHB.PerformanceControlManualValue, out2 => #PerformanceManualPrev)
   END_RUNG
   RUNG wire#powerrail
      N_Contact(operand := "CAN_Data_DB".InputData.CAN_ID_101h.ForcePerformanceControlSP, bit := #enForceMotorRpmSP)
      R_Coil( "DB_Application".ToHB.PerformanceControlManualMode )
   END_RUNG
   RUNG wire#powerrail
      P_Contact(operand := "CAN_Data_DB".InputData.CAN_ID_101h.ForceOilHeatingSP, bit := #epForceOilHeatingSP)
      wire#w4
      S_Coil( "DB_Application".ToHB.OilHeatingRegulatorManualMode )
   END_RUNG
   RUNG wire#powerrail
      Contact( "CAN_Data_DB".InputData.CAN_ID_101h.ForceOilHeatingSP )
      { S7_Templates := "SrcType := Real" } NE_Contact(in1 := "CAN_Data_DB".InputData.CAN_ID_103h.OilHeatingSP, in2 := #OilHeatingManualPrev)
   END_RUNG wire#w4
   RUNG wire#w4
      Move(in := "CAN_Data_DB".InputData.CAN_ID_103h.OilHeatingSP, out1 => "DB_Application".ToHB.OilHeatingManualValue, out2 => #OilHeatingManualPrev)
   END_RUNG
   RUNG wire#powerrail
      N_Contact(operand := "CAN_Data_DB".InputData.CAN_ID_101h.ForceOilHeatingSP, bit := #enForceOilHeatingSP)
      R_Coil( "DB_Application".ToHB.OilHeatingRegulatorManualMode )
   END_RUNG
   RUNG wire#powerrail
      P_Contact(operand := "CAN_Data_DB".InputData.CAN_ID_101h.ForcePinchSP, bit := #epForcePinchSP)
      wire#w5
      S_Coil( "DB_Application".ToHB.PinchRegulatorManualMode )
   END_RUNG
   RUNG wire#powerrail
      Contact( "CAN_Data_DB".InputData.CAN_ID_101h.ForcePinchSP )
      { S7_Templates := "SrcType := Real" } NE_Contact(in1 := "CAN_Data_DB".InputData.CAN_ID_104h.PinchSP, in2 := #PinchManualPrev)
   END_RUNG wire#w5
   RUNG wire#w5
      Move(in := "CAN_Data_DB".InputData.CAN_ID_104h.PinchSP, out1 => "DB_Application".ToHB.PinchManualValue, out2 => #PinchManualPrev)
   END_RUNG
   RUNG wire#powerrail
      N_Contact(operand := "CAN_Data_DB".InputData.CAN_ID_101h.ForcePinchSP, bit := #enForcePinchSP)
      R_Coil( "DB_Application".ToHB.PinchRegulatorManualMode )
   END_RUNG
   RUNG wire#powerrail
      P_Contact(operand := "CAN_Data_DB".InputData.CAN_ID_101h.ForceSuperheatSP, bit := #epForceSuperheatSP)
      wire#w6
      S_Coil( "DB_Application".ToHB.SuperheatManualMode )
   END_RUNG
   RUNG wire#powerrail
      Contact( "CAN_Data_DB".InputData.CAN_ID_101h.ForceSuperheatSP )
      { S7_Templates := "SrcType := Real" } NE_Contact(in1 := "CAN_Data_DB".InputData.CAN_ID_102h.SuperheatSP, in2 := #SuperheatManualPrev)
   END_RUNG wire#w6
   RUNG wire#w6
      Move(in := "CAN_Data_DB".InputData.CAN_ID_102h.SuperheatSP, out1 => "DB_Application".ToHB.SuperheatManualValue, out2 => #SuperheatManualPrev)
   END_RUNG
   RUNG wire#powerrail
      N_Contact(operand := "CAN_Data_DB".InputData.CAN_ID_101h.ForceSuperheatSP, bit := #enForceSuperheatSP)
      R_Coil( "DB_Application".ToHB.SuperheatManualMode )
   END_RUNG
   // the same network as SCL:
   #_w1 := "CAN_Data_DB".InputData.CAN_ID_101h.ForceExpansionValveSP AND NOT #epForceExpansionValveSP;   // rising edge of "CAN_Data_DB".InputData.CAN_ID_101h.ForceExpansionValveSP
   #epForceExpansionValveSP := "CAN_Data_DB".InputData.CAN_ID_101h.ForceExpansionValveSP;
   IF #_w1 OR ("CAN_Data_DB".InputData.CAN_ID_101h.ForceExpansionValveSP AND ("CAN_Data_DB".InputData.CAN_ID_104h.ExpansionValveSP <> #ExpansionManualPrev)) THEN
       "DB_Application".ToHB.ExpansionValveRegulatorManualMode := TRUE;
       "DB_Application".ToHB.ExpansionValveManualValue := "CAN_Data_DB".InputData.CAN_ID_104h.ExpansionValveSP;
       #ExpansionManualPrev := "CAN_Data_DB".InputData.CAN_ID_104h.ExpansionValveSP;
   END_IF;
   #_w2 := NOT "CAN_Data_DB".InputData.CAN_ID_101h.ForceExpansionValveSP AND #enForceExpansionValveSP;   // falling edge of "CAN_Data_DB".InputData.CAN_ID_101h.ForceExpansionValveSP
   #enForceExpansionValveSP := "CAN_Data_DB".InputData.CAN_ID_101h.ForceExpansionValveSP;
   IF #_w2 THEN "DB_Application".ToHB.ExpansionValveRegulatorManualMode := FALSE; END_IF;
   #_w3 := "CAN_Data_DB".InputData.CAN_ID_101h.ForceHeatSinkOutSP AND NOT #epForceHeatSinkOutSP;   // rising edge of "CAN_Data_DB".InputData.CAN_ID_101h.ForceHeatSinkOutSP
   #epForceHeatSinkOutSP := "CAN_Data_DB".InputData.CAN_ID_101h.ForceHeatSinkOutSP;
   IF #_w3 OR ("CAN_Data_DB".InputData.CAN_ID_101h.ForceHeatSinkOutSP AND ("CAN_Data_DB".InputData.CAN_ID_102h.HeatSinkOutSP <> #HeatSinkManualPrev)) THEN
       "DB_Application".ToHB.HeatSinkOutManualMode := TRUE;
       "DB_Application".ToHB.HeatSinkOutManualValue := "CAN_Data_DB".InputData.CAN_ID_102h.HeatSinkOutSP;
       #HeatSinkManualPrev := "CAN_Data_DB".InputData.CAN_ID_102h.HeatSinkOutSP;
   END_IF;
   #_w4 := NOT "CAN_Data_DB".InputData.CAN_ID_101h.ForceHeatSinkOutSP AND #enForceHeatSinkOutSP;   // falling edge of "CAN_Data_DB".InputData.CAN_ID_101h.ForceHeatSinkOutSP
   #enForceHeatSinkOutSP := "CAN_Data_DB".InputData.CAN_ID_101h.ForceHeatSinkOutSP;
   IF #_w4 THEN "DB_Application".ToHB.HeatSinkOutManualMode := FALSE; END_IF;
   #_w5 := "CAN_Data_DB".InputData.CAN_ID_101h.ForcePerformanceControlSP AND NOT #epForceMotorRpmSP;   // rising edge of "CAN_Data_DB".InputData.CAN_ID_101h.ForcePerformanceControlSP
   #epForceMotorRpmSP := "CAN_Data_DB".InputData.CAN_ID_101h.ForcePerformanceControlSP;
   IF #_w5 OR ("CAN_Data_DB".InputData.CAN_ID_101h.ForcePerformanceControlSP AND ("CAN_Data_DB".InputData.CAN_ID_103h.PerformanceControlSP <> #PerformanceManualPrev)) THEN
       "DB_Application".ToHB.PerformanceControlManualMode := TRUE;
       "DB_Application".ToHB.PerformanceControlManualValue := "CAN_Data_DB".InputData.CAN_ID_103h.PerformanceControlSP;
       #PerformanceManualPrev := "CAN_Data_DB".InputData.CAN_ID_103h.PerformanceControlSP;
   END_IF;
   #_w6 := NOT "CAN_Data_DB".InputData.CAN_ID_101h.ForcePerformanceControlSP AND #enForceMotorRpmSP;   // falling edge of "CAN_Data_DB".InputData.CAN_ID_101h.ForcePerformanceControlSP
   #enForceMotorRpmSP := "CAN_Data_DB".InputData.CAN_ID_101h.ForcePerformanceControlSP;
   IF #_w6 THEN "DB_Application".ToHB.PerformanceControlManualMode := FALSE; END_IF;
   #_w7 := "CAN_Data_DB".InputData.CAN_ID_101h.ForceOilHeatingSP AND NOT #epForceOilHeatingSP;   // rising edge of "CAN_Data_DB".InputData.CAN_ID_101h.ForceOilHeatingSP
   #epForceOilHeatingSP := "CAN_Data_DB".InputData.CAN_ID_101h.ForceOilHeatingSP;
   IF #_w7 OR ("CAN_Data_DB".InputData.CAN_ID_101h.ForceOilHeatingSP AND ("CAN_Data_DB".InputData.CAN_ID_103h.OilHeatingSP <> #OilHeatingManualPrev)) THEN
       "DB_Application".ToHB.OilHeatingRegulatorManualMode := TRUE;
       "DB_Application".ToHB.OilHeatingManualValue := "CAN_Data_DB".InputData.CAN_ID_103h.OilHeatingSP;
       #OilHeatingManualPrev := "CAN_Data_DB".InputData.CAN_ID_103h.OilHeatingSP;
   END_IF;
   #_w8 := NOT "CAN_Data_DB".InputData.CAN_ID_101h.ForceOilHeatingSP AND #enForceOilHeatingSP;   // falling edge of "CAN_Data_DB".InputData.CAN_ID_101h.ForceOilHeatingSP
   #enForceOilHeatingSP := "CAN_Data_DB".InputData.CAN_ID_101h.ForceOilHeatingSP;
   IF #_w8 THEN "DB_Application".ToHB.OilHeatingRegulatorManualMode := FALSE; END_IF;
   #_w9 := "CAN_Data_DB".InputData.CAN_ID_101h.ForcePinchSP AND NOT #epForcePinchSP;   // rising edge of "CAN_Data_DB".InputData.CAN_ID_101h.ForcePinchSP
   #epForcePinchSP := "CAN_Data_DB".InputData.CAN_ID_101h.ForcePinchSP;
   IF #_w9 OR ("CAN_Data_DB".InputData.CAN_ID_101h.ForcePinchSP AND ("CAN_Data_DB".InputData.CAN_ID_104h.PinchSP <> #PinchManualPrev)) THEN
       "DB_Application".ToHB.PinchRegulatorManualMode := TRUE;
       "DB_Application".ToHB.PinchManualValue := "CAN_Data_DB".InputData.CAN_ID_104h.PinchSP;
       #PinchManualPrev := "CAN_Data_DB".InputData.CAN_ID_104h.PinchSP;
   END_IF;
   #_w10 := NOT "CAN_Data_DB".InputData.CAN_ID_101h.ForcePinchSP AND #enForcePinchSP;   // falling edge of "CAN_Data_DB".InputData.CAN_ID_101h.ForcePinchSP
   #enForcePinchSP := "CAN_Data_DB".InputData.CAN_ID_101h.ForcePinchSP;
   IF #_w10 THEN "DB_Application".ToHB.PinchRegulatorManualMode := FALSE; END_IF;
   #_w11 := "CAN_Data_DB".InputData.CAN_ID_101h.ForceSuperheatSP AND NOT #epForceSuperheatSP;   // rising edge of "CAN_Data_DB".InputData.CAN_ID_101h.ForceSuperheatSP
   #epForceSuperheatSP := "CAN_Data_DB".InputData.CAN_ID_101h.ForceSuperheatSP;
   IF #_w11 OR ("CAN_Data_DB".InputData.CAN_ID_101h.ForceSuperheatSP AND ("CAN_Data_DB".InputData.CAN_ID_102h.SuperheatSP <> #SuperheatManualPrev)) THEN
       "DB_Application".ToHB.SuperheatManualMode := TRUE;
       "DB_Application".ToHB.SuperheatManualValue := "CAN_Data_DB".InputData.CAN_ID_102h.SuperheatSP;
       #SuperheatManualPrev := "CAN_Data_DB".InputData.CAN_ID_102h.SuperheatSP;
   END_IF;
   #_w12 := NOT "CAN_Data_DB".InputData.CAN_ID_101h.ForceSuperheatSP AND #enForceSuperheatSP;   // falling edge of "CAN_Data_DB".InputData.CAN_ID_101h.ForceSuperheatSP
   #enForceSuperheatSP := "CAN_Data_DB".InputData.CAN_ID_101h.ForceSuperheatSP;
   IF #_w12 THEN "DB_Application".ToHB.SuperheatManualMode := FALSE; END_IF;
END_REGION

REGION Network 3: Start request
   // PumaSystemReady: Puma is ok
   // Clearance: Puma and the Test Support System are ok.
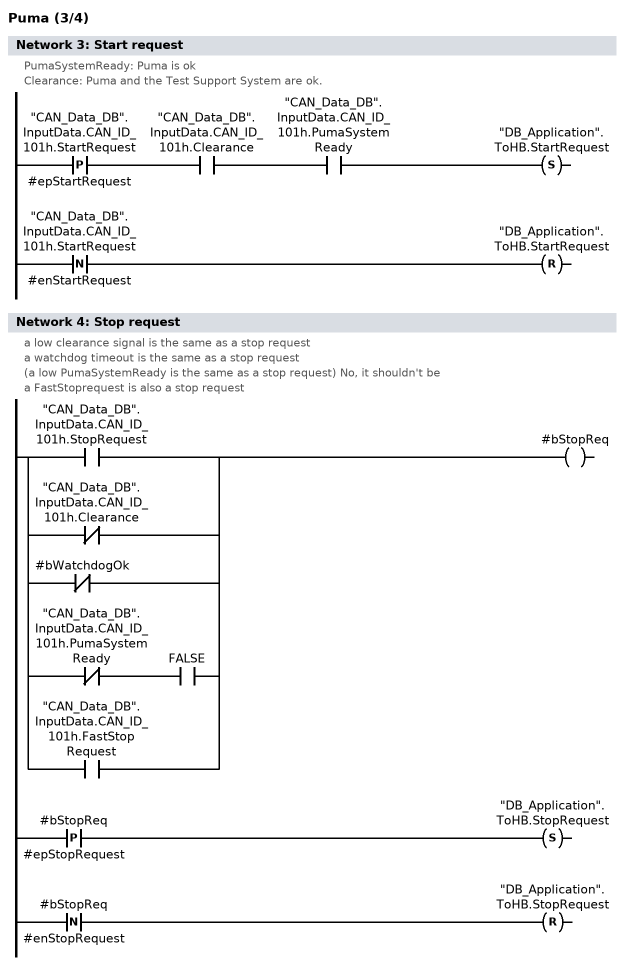
   RUNG wire#powerrail
      P_Contact(operand := "CAN_Data_DB".InputData.CAN_ID_101h.StartRequest, bit := #epStartRequest)
      Contact( "CAN_Data_DB".InputData.CAN_ID_101h.Clearance )
      Contact( "CAN_Data_DB".InputData.CAN_ID_101h.PumaSystemReady )
      S_Coil( "DB_Application".ToHB.StartRequest )
   END_RUNG
   RUNG wire#powerrail
      N_Contact(operand := "CAN_Data_DB".InputData.CAN_ID_101h.StartRequest, bit := #enStartRequest)
      R_Coil( "DB_Application".ToHB.StartRequest )
   END_RUNG
   // the same network as SCL:
   #_w1 := "CAN_Data_DB".InputData.CAN_ID_101h.StartRequest AND NOT #epStartRequest;   // rising edge of "CAN_Data_DB".InputData.CAN_ID_101h.StartRequest
   #epStartRequest := "CAN_Data_DB".InputData.CAN_ID_101h.StartRequest;
   IF #_w1 AND "CAN_Data_DB".InputData.CAN_ID_101h.Clearance AND "CAN_Data_DB".InputData.CAN_ID_101h.PumaSystemReady THEN
       "DB_Application".ToHB.StartRequest := TRUE;
   END_IF;
   #_w2 := NOT "CAN_Data_DB".InputData.CAN_ID_101h.StartRequest AND #enStartRequest;   // falling edge of "CAN_Data_DB".InputData.CAN_ID_101h.StartRequest
   #enStartRequest := "CAN_Data_DB".InputData.CAN_ID_101h.StartRequest;
   IF #_w2 THEN "DB_Application".ToHB.StartRequest := FALSE; END_IF;
END_REGION

REGION Network 4: Stop request
   // a low clearance signal is the same as a stop request
   // a watchdog timeout is the same as a stop request
   // (a low PumaSystemReady is the same as a stop request) No, it shouldn't be
   // a FastStoprequest is also a stop request
   RUNG wire#powerrail
      Contact( "CAN_Data_DB".InputData.CAN_ID_101h.StopRequest )
      wire#w1
      Coil( #bStopReq )
   END_RUNG
   RUNG wire#powerrail
      I_Contact( "CAN_Data_DB".InputData.CAN_ID_101h.Clearance )
   END_RUNG wire#w1
   RUNG wire#powerrail
      I_Contact( #bWatchdogOk )
   END_RUNG wire#w1
   RUNG wire#powerrail
      I_Contact( "CAN_Data_DB".InputData.CAN_ID_101h.PumaSystemReady )
      Contact( FALSE )
   END_RUNG wire#w1
   RUNG wire#powerrail
      Contact( "CAN_Data_DB".InputData.CAN_ID_101h.FastStopRequest )
   END_RUNG wire#w1
   RUNG wire#powerrail
      P_Contact(operand := #bStopReq, bit := #epStopRequest)
      S_Coil( "DB_Application".ToHB.StopRequest )
   END_RUNG
   RUNG wire#powerrail
      N_Contact(operand := #bStopReq, bit := #enStopRequest)
      R_Coil( "DB_Application".ToHB.StopRequest )
   END_RUNG
   // the same network as SCL:
   #bStopReq := "CAN_Data_DB".InputData.CAN_ID_101h.StopRequest OR NOT "CAN_Data_DB".InputData.CAN_ID_101h.Clearance OR NOT #bWatchdogOk OR (NOT "CAN_Data_DB".InputData.CAN_ID_101h.PumaSystemReady AND FALSE) OR "CAN_Data_DB".InputData.CAN_ID_101h.FastStopRequest;
   #_w1 := #bStopReq AND NOT #epStopRequest;   // rising edge of #bStopReq
   #epStopRequest := #bStopReq;
   IF #_w1 THEN "DB_Application".ToHB.StopRequest := TRUE; END_IF;
   #_w2 := NOT #bStopReq AND #enStopRequest;   // falling edge of #bStopReq
   #enStopRequest := #bStopReq;
   IF #_w2 THEN "DB_Application".ToHB.StopRequest := FALSE; END_IF;
END_REGION

REGION Network 5: Commands
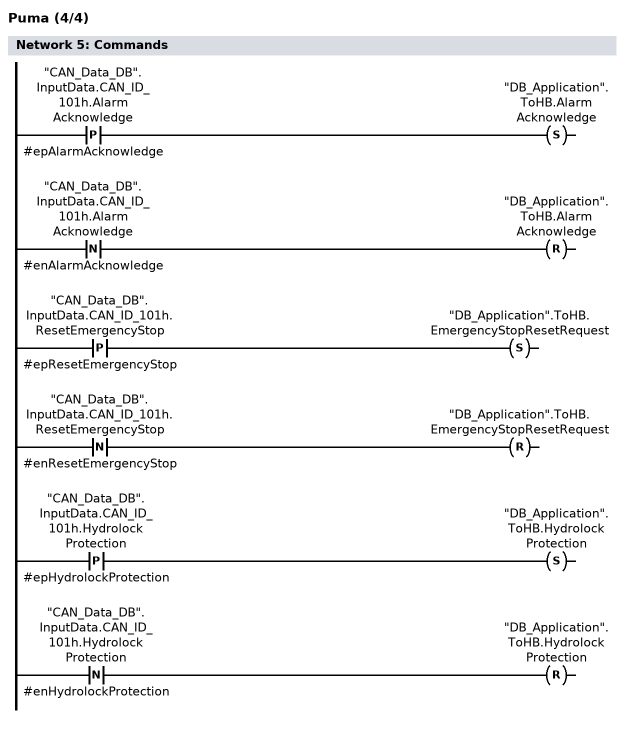
   RUNG wire#powerrail
      P_Contact(operand := "CAN_Data_DB".InputData.CAN_ID_101h.AlarmAcknowledge, bit := #epAlarmAcknowledge)
      S_Coil( "DB_Application".ToHB.AlarmAcknowledge )
   END_RUNG
   RUNG wire#powerrail
      N_Contact(operand := "CAN_Data_DB".InputData.CAN_ID_101h.AlarmAcknowledge, bit := #enAlarmAcknowledge)
      R_Coil( "DB_Application".ToHB.AlarmAcknowledge )
   END_RUNG
   RUNG wire#powerrail
      P_Contact(operand := "CAN_Data_DB".InputData.CAN_ID_101h.ResetEmergencyStop, bit := #epResetEmergencyStop)
      S_Coil( "DB_Application".ToHB.EmergencyStopResetRequest )
   END_RUNG
   RUNG wire#powerrail
      N_Contact(operand := "CAN_Data_DB".InputData.CAN_ID_101h.ResetEmergencyStop, bit := #enResetEmergencyStop)
      R_Coil( "DB_Application".ToHB.EmergencyStopResetRequest )
   END_RUNG
   RUNG wire#powerrail
      P_Contact(operand := "CAN_Data_DB".InputData.CAN_ID_101h.HydrolockProtection, bit := #epHydrolockProtection)
      S_Coil( "DB_Application".ToHB.HydrolockProtection )
   END_RUNG
   RUNG wire#powerrail
      N_Contact(operand := "CAN_Data_DB".InputData.CAN_ID_101h.HydrolockProtection, bit := #enHydrolockProtection)
      R_Coil( "DB_Application".ToHB.HydrolockProtection )
   END_RUNG
   // the same network as SCL:
   #_w1 := "CAN_Data_DB".InputData.CAN_ID_101h.AlarmAcknowledge AND NOT #epAlarmAcknowledge;   // rising edge of "CAN_Data_DB".InputData.CAN_ID_101h.AlarmAcknowledge
   #epAlarmAcknowledge := "CAN_Data_DB".InputData.CAN_ID_101h.AlarmAcknowledge;
   IF #_w1 THEN "DB_Application".ToHB.AlarmAcknowledge := TRUE; END_IF;
   #_w2 := NOT "CAN_Data_DB".InputData.CAN_ID_101h.AlarmAcknowledge AND #enAlarmAcknowledge;   // falling edge of "CAN_Data_DB".InputData.CAN_ID_101h.AlarmAcknowledge
   #enAlarmAcknowledge := "CAN_Data_DB".InputData.CAN_ID_101h.AlarmAcknowledge;
   IF #_w2 THEN "DB_Application".ToHB.AlarmAcknowledge := FALSE; END_IF;
   #_w3 := "CAN_Data_DB".InputData.CAN_ID_101h.ResetEmergencyStop AND NOT #epResetEmergencyStop;   // rising edge of "CAN_Data_DB".InputData.CAN_ID_101h.ResetEmergencyStop
   #epResetEmergencyStop := "CAN_Data_DB".InputData.CAN_ID_101h.ResetEmergencyStop;
   IF #_w3 THEN "DB_Application".ToHB.EmergencyStopResetRequest := TRUE; END_IF;
   #_w4 := NOT "CAN_Data_DB".InputData.CAN_ID_101h.ResetEmergencyStop AND #enResetEmergencyStop;   // falling edge of "CAN_Data_DB".InputData.CAN_ID_101h.ResetEmergencyStop
   #enResetEmergencyStop := "CAN_Data_DB".InputData.CAN_ID_101h.ResetEmergencyStop;
   IF #_w4 THEN "DB_Application".ToHB.EmergencyStopResetRequest := FALSE; END_IF;
   #_w5 := "CAN_Data_DB".InputData.CAN_ID_101h.HydrolockProtection AND NOT #epHydrolockProtection;   // rising edge of "CAN_Data_DB".InputData.CAN_ID_101h.HydrolockProtection
   #epHydrolockProtection := "CAN_Data_DB".InputData.CAN_ID_101h.HydrolockProtection;
   IF #_w5 THEN "DB_Application".ToHB.HydrolockProtection := TRUE; END_IF;
   #_w6 := NOT "CAN_Data_DB".InputData.CAN_ID_101h.HydrolockProtection AND #enHydrolockProtection;   // falling edge of "CAN_Data_DB".InputData.CAN_ID_101h.HydrolockProtection
   #enHydrolockProtection := "CAN_Data_DB".InputData.CAN_ID_101h.HydrolockProtection;
   IF #_w6 THEN "DB_Application".ToHB.HydrolockProtection := FALSE; END_IF;
END_REGION
END_FUNCTION_BLOCK

FUNCTION_BLOCK "fbHeartbeatCount2"
{ S7_Optimized_Access := 'TRUE' }
VERSION : 0.1
   VAR_INPUT 
      bEnable : Bool;   // 1 = run watchdog, 0 = do not run
      nLocalCount : UInt;
      nRemoteCount : UInt;
   END_VAR

   VAR_OUTPUT 
      bOk : Bool;   // Comm ok
   END_VAR

   VAR_IN_OUT 
      sTag : "stHeartbeatCount2";
   END_VAR

   VAR 
      Timeout {InstructionName := 'TON_TIME'; LibVersion := '1.0'; S7_SetPoint := 'False'} : TON_TIME;
      nRemoteCountPrev { S7_SetPoint := 'True'} : UInt := 0;
      Enabled { S7_SetPoint := 'True'} : Bool;
   END_VAR


BEGIN
	// fbHeartbeatCount2 - communications monitoring
	// Monitor a count for liveness. If it does not change within the timeout, it goes to error state
	// Include the local count here so it gets copied up to the HMI too for operator awareness.
	
	// Copy inputs to tag
	#sTag.nRemoteCount := #nRemoteCount;
	#sTag.nLocalCount := #nLocalCount;
	
	// Enable
	#Enabled := #bEnable AND #sTag.bEnable;
	
	// Timeout
	#Timeout(IN := (#sTag.nState = 2), PT := #sTag.tTimeout);
	
	// States
	CASE #sTag.nState OF
	    0: // Idle
	        #sTag.bOk := TRUE;
	        IF #Enabled = TRUE THEN
	            #sTag.nState := 1;
	        END_IF;
	    1: // Update
	        #nRemoteCountPrev := #nRemoteCount;
	        IF #Enabled = FALSE THEN
	            #sTag.nState := 0;
	        ELSE
	            #sTag.nState := 2;
	        END_IF;
	    2: // Wait
	        IF #nRemoteCount <> #nRemoteCountPrev THEN
	            // Pong
	            #sTag.bOk := TRUE;
	            #sTag.nState := 1;
	        ELSIF #Timeout.Q = TRUE THEN
	            #sTag.bOk := FALSE;
	            #sTag.nState := 1;
	        ELSIF #Enabled = FALSE THEN
	            #sTag.nState := 0;
	        END_IF;
	        
	END_CASE;
	
	// Local outputs
	#bOk := #sTag.bOk;
	
	
	
END_FUNCTION_BLOCK

FUNCTION_BLOCK "Customer"   // FB3, LAD
TITLE = Combine signals from Customer into DB_Application
{ S7_Optimized_Access := 'TRUE' }
AUTHOR : Heaten
VERSION : 0.1
// stored: AutoNumber true, IsIECCheckEnabled false, IsRetainMemResEnabled false, MemoryReserve 100, SetENOAutomatically false, UDAEnableTagReadback false
   VAR
      Watchdog { S7_SetPoint := 'True'} : "fbHeartbeatCount2";
      epStartRequest { S7_SetPoint := 'True'} : Bool;
      enStartRequest : Bool;
      epStopRequest : Bool;
      enStopRequest : Bool;
      epAlarmAcknowledge : Bool;
      enAlarmAcknowledge : Bool;
      epResetEmergencyStop : Bool;
      enResetEmergencyStop : Bool;
      SetpointPrev : Real;
      RegulationTargetPrev : Int;
      HCV812Cmd : Real;   // TEMPORARY
      HCV815Cmd : Real;   // TEMPORARY
      HCV818Cmd : Real;   // TEMPORARY
      HCV821Cmd : Real;   // TEMPORARY
   END_VAR
   VAR_TEMP
      bWatchdogOk : Bool;
      bStopReq : Bool;
      fDummy : Real;
      iDummy : Int;
   END_VAR
   VAR_TEMP   // added for the SCL form of the ladder/FBD networks
      _w1 : Bool;
      _w2 : Bool;
      _w3 : Bool;
      _w4 : Bool;
   END_VAR
BEGIN

REGION Network 1: Map IO tags to DBs
   // When using S7 communication this mapping is not necessary
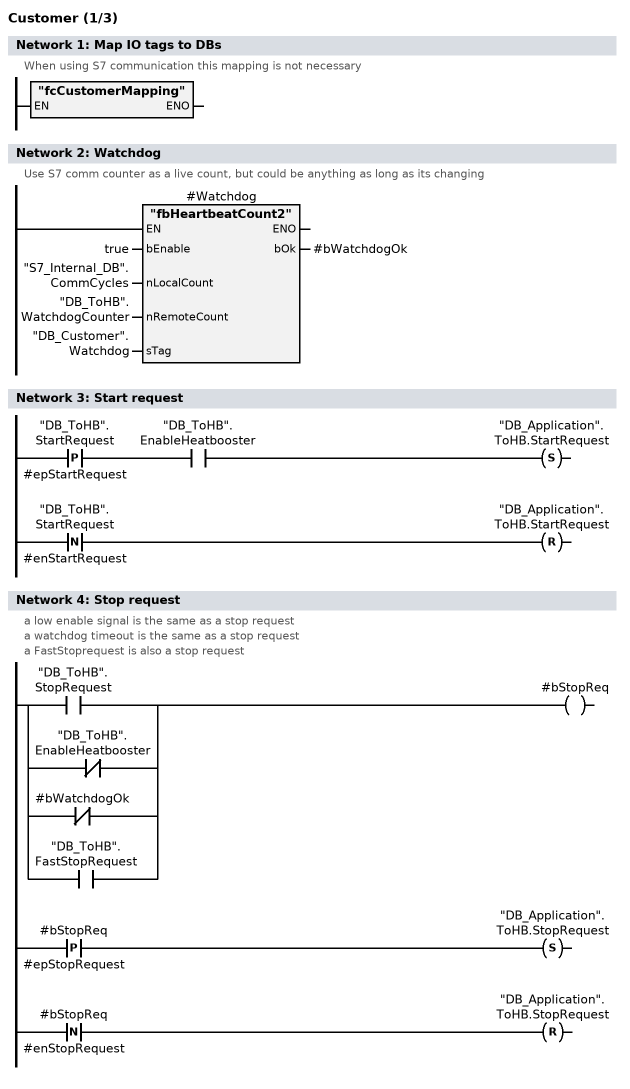
   RUNG wire#powerrail
      "fcCustomerMapping"()
   END_RUNG
   // the same network as SCL:
   "fcCustomerMapping"();
END_REGION

